// TwinCAT 3 PLC project Untitled1
// ProgramVersion: 3.1.4023.0
// libraries:
//   Tc2_EtherCAT, * (Beckhoff Automation GmbH)
//   Tc2_ModbusSrv, * (Beckhoff Automation GmbH)
//   Tc2_Standard, * (Beckhoff Automation GmbH)
//   Tc2_System, * (Beckhoff Automation GmbH)
//   Tc3_Module, * (Beckhoff Automation GmbH)
//   VisuDialogs, * (System)
//   BASIC,3.31,OSCAT
//   VisuSymbols,3.5.10.0,System
// project tree:
//   / Control.TcTTO, GlobalTextList.TcGTLO, Meter.TcTTO, PlcTask_1.TcTTO, Visualization Manager.TcVMO (not stored), VISU_TASK.TcTTO
//   DUTs/ CONVERTER.TcDUT
//   FUNC/ AVG_3.TcPOU, BYTE_UNION.TcPOU (not stored)
//   GVLs/ GVL_PM_CONFIG.TcGVL, GVL_GUI.TcGVL, GVL_HANDLER.TcGVL, GVL_POWERMETER.TcGVL, GVL_CONVERTERS_COMMON.TcGVL, GVL_CONV_COMMS.TcGVL, GVL_PLANT_DEF.TcGVL, GVL_P_CONTROL.TcGVL, GVL_Q_CONTROL.TcGVL, Meter_board_str.TcDUT
//   POUs/ BYTE_UNION.TcPOU, MAIN.TcPOU
//   POUs/CONTROL/ PI_BLOCK.TcPOU
//   POUs/CONVERTERS/ CONVERTERS_COMMS.TcPOU, Modbus_mapping.TcPOU, nN_coeff_calculation.TcPOU
//   POUs/EXTERNAL_COMMS/ Modbus_map.TcDUT
//   POUs/HANDLER_PARAM/ Data_transforming.TcPOU, Data_transform_float32.TcPOU, Data_transform_int64.TcPOU, MB_MAP_VARS_ENUM.TcTLEO, Parameters_handler.TcPOU, ReadWrite_Enum.TcDUT
//   POUs/METERING/ Analyzers.TcPOU, FB_EL3453_handling.TcPOU, METER_BOARD_CFG.TcPOU, METER_EL3453_CFG.TcPOU
//   POUs/P CONTROL/ Min_P_calculation.TcPOU, P_control_global.TcPOU, P_feedback_calculation.TcPOU
//   POUs/Q CONTROL/ Q_control_global.TcPOU, Q_ramp_module.TcPOU
//   POUs/VISU_HANDLER/ GUI_logic.TcPOU
//   VISUs/00_Main/ Main.TcVIS, Main_GUI.TcVIS
//   VISUs/01_P_control/ P_controller.TcVIS, P_min_indicator.TcTLO
//   VISUs/02_Q_control/ Q_controller.TcVIS
//   VISUs/03_Converters/ Conv_handling.TcVIS
//   VISUs/04_Powermeter/ M_board_status.TcTLO, PM_config.TcVIS
// real-time tasks:
//   TASK PlcTask: cycle T#5ms, priority 20, ADS port 350
//   TASK Control: cycle T#5ms, priority 1, ADS port 351
//   TASK Meter: cycle T#1ms, priority 2, ADS port 352
//   TASK VISU_TASK: cycle T#200000us, priority 30, ADS port 354
// I/O:
//   DEVICE Device 1 (EtherCAT) (disabled), AmsNetId 192.168.222.1.2.1
//     Term 1 (EK1200) [EK1200-7000 EtherCAT Power supply (1,5A E-Bus)] (disabled)
//       Term 4 (EL1259) [EL1259 8Ch. Dig Input 24V/8Ch. Dig. Output 24V with Multi-Time-Stamp] (disabled)
//       Term 5 (EL3453) [EL3453 3Ch. Power Measuring] (disabled)
//       Term 3 (EL9011) [EL9011 End Terminal]
// variable links:
//   Untitled1/Untitled1 Instance <-> Device 1 (EtherCAT)/Term 1 (EK1200)/Term 5 (EL3453)
//     Meter Inputs/GVL_POWERMETER.M_board_Freq_Hz <-> Total Basic/Frequency
//     Meter Inputs/GVL_POWERMETER.M_board_I_L1_angle <-> Total System Angles/Current Angle L1
//     Meter Inputs/GVL_POWERMETER.M_board_I_L2_angle <-> Total System Angles/Current Angle L2
//     Meter Inputs/GVL_POWERMETER.M_board_I_L3_angle <-> Total System Angles/Current Angle L3
//     Meter Inputs/GVL_POWERMETER.M_board_P_L1_kW <-> L1 Power/Active Power
//     Meter Inputs/GVL_POWERMETER.M_board_P_L2_kW <-> L2 Power/Active Power
//     Meter Inputs/GVL_POWERMETER.M_board_P_L3_kW <-> L3 Power/Active Power
//     Meter Inputs/GVL_POWERMETER.M_board_P_kW <-> Total Active Reduced/Active Power
//     Meter Inputs/GVL_POWERMETER.M_board_Q_L1_kVAr <-> L1 Power/Reactive Power
//     Meter Inputs/GVL_POWERMETER.M_board_Q_L2_kVAr <-> L2 Power/Reactive Power
//     Meter Inputs/GVL_POWERMETER.M_board_Q_L3_kVAr <-> L3 Power/Reactive Power
//     Meter Inputs/GVL_POWERMETER.M_board_Q_kVAr <-> Total Reactive Reduced/Reactive Power
//     Meter Inputs/GVL_POWERMETER.M_board_S_L1_kVA <-> L1 Power/Apparent Power
//     Meter Inputs/GVL_POWERMETER.M_board_S_L2_kVA <-> L2 Power/Apparent Power
//     Meter Inputs/GVL_POWERMETER.M_board_S_L3_kVA <-> L3 Power/Apparent Power
//     Meter Inputs/GVL_POWERMETER.M_board_S_kVA <-> Total Apparent Reduced/Apparent Power
//     Meter Inputs/GVL_POWERMETER.M_board_V_L1L2_Volt <-> Total L-L Voltages/L1-L2 Voltage
//     Meter Inputs/GVL_POWERMETER.M_board_V_L2L3_Volt <-> Total L-L Voltages/L2-L3 Voltage
//     Meter Inputs/GVL_POWERMETER.M_board_V_L3L1_Volt <-> Total L-L Voltages/L3-L1 Voltage
//     Meter Inputs/GVL_POWERMETER.M_board_V_L1L2_angle <-> Total System Angles/Voltage Angle L1L2
//     Meter Inputs/GVL_POWERMETER.M_board_V_L1L3_angle <-> Total System Angles/Voltage Angle L1L3
//     Meter Inputs/GVL_POWERMETER.M_board_V_L1N_Volt <-> L1 Basic/Voltage
//     Meter Inputs/GVL_POWERMETER.M_board_V_L2N_Volt <-> L2 Basic/Voltage
//     Meter Inputs/GVL_POWERMETER.M_board_V_L3N_Volt <-> L3 Basic/Voltage
//     Meter Inputs/GVL_POWERMETER.M_board_cos_phi <-> Total Basic/Power Factor
//     Meter Inputs/GVL_POWERMETER.M_board_cos_phi_L1 <-> L1 Power/Power Factor
//     Meter Inputs/GVL_POWERMETER.M_board_cos_phi_L2 <-> L2 Power/Power Factor
//     Meter Inputs/GVL_POWERMETER.M_board_cos_phi_L3 <-> L3 Power/Power Factor
//     PlcTask_1 Inputs/GVL_POWERMETER.M_board_Meter_status <-> InfoData/State

CONFIGURATION Untitled1
    RESOURCE PLC ON TwinCAT3
        TASK Control(INTERVAL := T#5ms, PRIORITY := 1);
        TASK Meter(INTERVAL := T#1ms, PRIORITY := 2);
        TASK PlcTask_1(INTERVAL := T#5ms, PRIORITY := 20);
        TASK VISU_TASK(INTERVAL := T#200000us, PRIORITY := 30);
        PROGRAM Q_control_global WITH Control : Q_control_global;
        PROGRAM P_control_global WITH Control : P_control_global;
        PROGRAM Analyzers WITH Meter : Analyzers;
        PROGRAM MAIN WITH PlcTask_1 : MAIN;
        PROGRAM VisuElems_Visu_Prg WITH VISU_TASK : VisuElems.Visu_Prg;
    END_RESOURCE
END_CONFIGURATION

// ---- DUTs/CONVERTER.TcDUT
TYPE CONVERTER :
STRUCT
	ReadRegs_INV: FB_MBReadRegs;
	WriteRegs_INV: FB_MBWriteRegs;
	
	Capacity: REAL:= 1000;				//Snominal from inverter in kVA
	IP: STRING(15):= '192.168.1.254';
	Port: UINT:= 502;					//Modbus port
	UnitID: BYTE:= 1;					//Modbus ID if necessary
	LengthRead: WORD:= 10;				//Amount of registers read from modbus
	LengthWrite: WORD:= 10;				//Amount of registers written via modbus
	InitAdressRead: WORD:= 7000;
	InitAdressWrite: WORD:= 8000;
	cbLenght: UDINT:= 2;
	READING: ARRAY [1..5] OF WORD;
    bReadBusy: BOOL;
    bReadError: BOOL;
    nReadErrorId: UDINT;
    nReadCount: UDINT;
	bWriteBusy: BOOL;
    bWriteError: BOOL;
    nWriteErrorId: UDINT;
    nWriteCount: UDINT;
	WRITING: ARRAY [1..7] OF WORD;
	ErrorCount: UDINT:= 0;
END_STRUCT
END_TYPE

// ---- GVLs/Meter_board_str.TcDUT
TYPE Meter_board_str :
STRUCT
	
	//Single-phase electrical parameters in engineering units
	P_L1_kW:			REAL;
	P_L2_kW:			REAL;
	P_L3_kW:			REAL;
	Q_L1_kVAr:			REAL;
	Q_L2_kVAr:			REAL;
	Q_L3_kVAr:			REAL;
	S_L1_kVA:			REAL;
	S_L2_kVA:			REAL;
	S_L3_kVA:			REAL;
	cos_phi_L1:			REAL;
	cos_phi_L2:			REAL;
	cos_phi_L3:			REAL;
	V_L1N_Volt:			REAL;
	V_L2N_Volt:			REAL;
	V_L3N_Volt:			REAL;

	//Three-phase electrical parameters in engineering units
	P_kW:				REAL;
	Q_kVAr:				REAL;
	S_kVA:				REAL;
	Freq_Hz:			REAL;
	cos_phi:			REAL;
	V_L1L2_Volt:		REAL;
	V_L2L3_Volt:		REAL;
	V_L3L1_Volt:		REAL;
	I_L1_angle:			REAL;
	I_L2_angle:			REAL;
	I_L3_angle:			REAL;
	V_L1L2_angle:		REAL;
	V_L1L3_angle:		REAL;
	
END_STRUCT
END_TYPE

// ---- POUs/EXTERNAL_COMMS/Modbus_map.TcDUT
{attribute 'qualified_only'}
{attribute 'strict'}
TYPE Modbus_map :
(
	enum_member := 0
);
END_TYPE

// ---- POUs/HANDLER_PARAM/MB_MAP_VARS_ENUM.TcTLEO
TYPE MB_MAP_VARS_ENUM :
(
	Plant_S_nom:= 0,
	Plant_V_nom:= 2,
	Plant_f_nom:= 4,
	N_converters:= 20,
	nN_converters:= 21,
	Control_conv_0:= 22,
	Control_conv_1:= 23,
	Control_conv_2:= 24,
	Control_conv_3:= 25,
	Control_conv_4:= 26,
	Control_conv_5:= 27,
	Control_conv_6:= 28,
	Control_conv_7:= 29,
	Control_conv_8:= 30,
	Control_conv_9:= 31,
	Control_conv_10:= 32,
	Control_conv_11:= 33,
	Control_conv_12:= 34,
	Control_conv_13:= 35,
	Control_conv_14:= 36,
	Control_conv_15:= 37,
	Control_conv_16:= 38,
	Control_conv_17:= 39,
	Control_conv_18:= 40,
	Control_conv_19:= 41,
	Control_conv_20:= 42,
	Control_conv_21:= 43,
	Control_conv_22:= 44,
	Control_conv_23:= 45,
	Control_conv_24:= 46,
	Control_conv_25:= 47,
	P_loop:= 300,
	P_reference:= 301,
	P_feedback:= 302,
	P_output:= 303,
	P_kp:= 304,
	P_kp_min:= 305,
	P_ti:= 306,
	P_high:= 307,
	P_low:= 308,
	P_invert:= 309,
	P_safety:= 310,
	P_min_charge:= 311,
	Q_loop:= 500,
	Q_reference:= 501,
	Q_feedback:= 502,
	Q_output:= 503,
	Q_kp:= 504,
	Q_kp_min:= 505,
	Q_ti:= 506,
	Q_high:= 507,
	Q_low:= 508,
	Q_invert:= 509,
	Q_safety:= 510,
	Ramp_enable:= 511,
	Time_span:= 512,
	R_up_value:= 513,
	R_down_value:= 514,
	R_units:= 515,
	P_L1_kW:= 1000,
	P_L2_kW:= 1002,
	P_L3_kW:= 1004,
	Q_L1_kVAr:= 1006,
	Q_L2_kVAr:= 1008,
	Q_L3_kVAr:= 1010,
	S_L1_kVA:= 1012,
	S_L2_kVA:= 1014,
	S_L3_kVA:= 1016,
	cos_phi_L1:= 1018,
	cos_phi_L2:= 1020,
	cos_phi_L3:= 1022,
	V_L1N_Volt:= 1024,
	V_L2N_Volt:= 1026,
	V_L3N_Volt:= 1028,
	P_tot_kW:= 1030,
	Q_tot_kVAr:= 1032,
	S_tot_kVA:= 1034,
	Freq_Hz:= 1036,
	cos_phi:= 1038,
	V_L1L2_Volt:= 1040,
	V_L2L3_Volt:= 1042,
	V_L3L1_Volt:= 1044,
	I_L1_angle:= 1046,
	I_L2_angle:= 1048,
	I_L3_angle:= 1050,
	V_L1L2_angle:= 1052,
	V_L1L3_angle:= 1054,
	V_phase_avg_Volt:= 1080,
	V_line_avg_Volt:= 1082,
	P_L1_pu:= 1084,
	P_L2_pu:= 1086,
	P_L3_pu:= 1088,
	Q_L1_pu:= 1090,
	Q_L2_pu:= 1092,
	Q_L3_pu:= 1094,
	S_L1_pu:= 1096,
	S_L2_pu:= 1098,
	S_L3_pu:= 1100,
	P_tot_pu:= 1102,
	Q_tot_pu:= 1104,
	S_tot_pu:= 1106,
	V_phase_avg_pu:= 1108,
	V_line_avg_pu:= 1110,
	Meter_status:= 1130,
	Lost_comms_enable:= 1131,
	Active_er_pos_kWh:= 1200,
	Active_er_neg_kWh:= 1204,
	Active_er_tot_kWh:= 1208,
	React_er_pos_kVArh:= 1212,
	React_er_neg_kVArh:= 1216,
	React_er_tot_kVArh:= 1220,
	Energies_reset:= 1224,
	V_ratio_RS:= 1300,
	V_ratio_ST:= 1302,
	V_ratio_TR:= 1304,
	I_ratio_R:=	1306,
	I_ratio_S:=	1308,
	I_ratio_T:=	1310

);
END_TYPE

// ---- POUs/HANDLER_PARAM/ReadWrite_Enum.TcDUT

TYPE ReadWrite_Enum :
(
	R_O := 0,
	R_W := 1
);
END_TYPE

// ---- GVLs/GVL_PM_CONFIG.TcGVL
{attribute 'qualified_only'}
VAR_GLOBAL
	
	//Variables needed to be in the data handling for the CoE analyzers boards configuration
	Device_Type_Index				: INT;
	Nominal_Voltage 				: REAL;
	Nominal_Frequency 				: REAL;
	Measurement_freq_range			: REAL;
	Current_trafo_dly_L1 			: REAL;			// Set variable for Current transformer delay L1	
	Current_trafo_dly_L2 			: REAL;			// Set variable for Current transformer delay L2
	Current_trafo_dly_L3 			: REAL;			// Set variable for Current transformer delay L3
	Current_trafo_range_L1 			: UDINT;		// Set variable for Current transformer range L1
	Current_trafo_range_L2 			: UDINT;		// Set variable for Current transformer range L2
	Current_trafo_range_L3 			: UDINT;		// Set variable for Current transformer range L3
	Voltage_Guard_Min_Error_L1		: REAL;			// Set variable for Voltage min error L1
	Voltage_Guard_Min_Error_L2		: REAL;			// Set variable for Voltage min error L2
	Voltage_Guard_Min_Error_L3		: REAL;			// Set variable for Voltage min error L3
	Voltage_Guard_Min_Warning_L1	: REAL;			// Set variable for Voltage min warning L1
	Voltage_Guard_Min_Warning_L2	: REAL;			// Set variable for Voltage min warning L2
	Voltage_Guard_Min_Warning_L3	: REAL;			// Set variable for Voltage min warning L3
	Voltage_Guard_Max_Warning_L1	: REAL;			// Set variable for Voltage max warning L1
	Voltage_Guard_Max_Warning_L2	: REAL;			// Set variable for Voltage max warning L2
	Voltage_Guard_Max_Warning_L3	: REAL;			// Set variable for Voltage max warning L3
	Voltage_Guard_Max_Error_L1		: REAL;			// Set variable for Voltage max error L1
	Voltage_Guard_Max_Error_L2		: REAL;			// Set variable for Voltage max error L2
	Voltage_Guard_Max_Error_L3		: REAL;			// Set variable for Voltage max error L3

	NetID_EL3XXX 		AT %I*	: AMSNETID ;
	SlaveID_EL3XXX 		AT %I*	: WORD ;
	 	
	NetID_EL3XXX_2 		AT %I*	: AMSNETID ;
	SlaveID_EL3XXX_2 	AT %I*	: WORD ;
END_VAR

VAR_GLOBAL PERSISTENT
	Current_trafo_rat_L1 			: REAL;			// Set variable for Current transformer ratio L1
	Current_trafo_rat_L2 			: REAL;			// Set variable for Current transformer ratio L2
	Current_trafo_rat_L3 			: REAL;			// Set variable for Current transformer ratio L3
	Voltage_trafo_rat_L1 			: REAL;			// Set variable for Voltage transformer ratio L1
	Voltage_trafo_rat_L2 			: REAL;			// Set variable for Voltage transformer ratio L2
	Voltage_trafo_rat_L3 			: REAL;			// Set variable for Voltage transformer ratio L3
END_VAR

// ---- GVLs/GVL_GUI.TcGVL
{attribute 'qualified_only'}
VAR_GLOBAL
	//Main GUI logic
	main_button_logic: 			BOOL:= TRUE;
	pcontrol_button_logic: 		BOOL:= FALSE;
	qcontrol_button_logic:		BOOL:= FALSE;
	conv_button_logic:			BOOL:= FALSE;
	meter_cfg_button_logic:		BOOL:= FALSE;
	
	frame_indic:				WORD:= 0;
	
	//P controller screen vars
	P_OL_sel_button:			BOOL:= FALSE;
	P_invert_button:			BOOL:= FALSE;
	
	//Q controller screen vars
	Q_OL_sel_button:			BOOL:= FALSE;
	Q_invert_button:			BOOL:= FALSE;
	
	//Converters screen
	Conv_online_button:			ARRAY [1..25] OF BOOL;
	Conv_on_off_button:			ARRAY [1..25] OF BOOL;
	Conv_n_mode_button:			ARRAY [1..25] OF BOOL;
END_VAR

// ---- GVLs/GVL_HANDLER.TcGVL
{attribute 'qualified_only'}
VAR_GLOBAL
	Init_vars:					BOOL; //initialization command
	Input_src:					bool:= false; //FALSE--> Via GUI, TRUE--> Via Modbus

	Modbus_srv_vars AT %MW0:	ARRAY [0..60000] OF WORD; //Variables for Modbus Server
	GUI_vars:					ARRAY [0..60000] OF REAL; //Variables for Web GUI
END_VAR

// ---- GVLs/GVL_POWERMETER.TcGVL
{attribute 'qualified_only'}
VAR_GLOBAL

	//Internal powermeter variables	
	Power_analyzer: 			Meter_board_str;
	Meter_comms_status: 		BOOL;
	
	//Internal calculated powermeter variables
		//Average voltages in engineering units
	V_phase_avg_Volt:			REAL;
	V_line_avg_Volt:			REAL;
		//Single-phase electrical parameters in p.u.
	P_L1_pu:					REAL;
	P_L2_pu:					REAL;
	P_L3_pu:					REAL;
	Q_L1_pu:					REAL;
	Q_L2_pu:					REAL;
	Q_L3_pu:					REAL;
	S_L1_pu:					REAL;
	S_L2_pu:					REAL;
	S_L3_pu:					REAL;
	V_L1N_pu:					REAL;
	V_L2N_pu:					REAL;
	V_L3N_pu:					REAL;
	I_L1_pu:					REAL;
	I_L2_pu:					REAL;
	I_L3_pu:					REAL;
		//Three-phase electrical parameters in p.u.
	P_pu:						REAL;
	Q_pu:						REAL;
	S_pu:						REAL;
		//Average voltages in engineering units
	V_phase_avg_pu:				REAL;
	V_line_avg_pu:				REAL;
	
	//Self-supply P variables
	P_min:						REAL; //Minimum P in p.u. of the system for PI feedback
	P_min_indicator:			WORD; //Minimum P indicator 0 --> L1; 1 --> L2; 2 --> L3

	//Enrgies handling & values
	Energies_reset:				BOOL:= FALSE;
	Active_er_neg_kWh: 			LINT:=0; //Active energy (three-phase) calculated if P_tot < 0
	Active_er_pos_kWh:			LINT:=0; //Active energy (three-phase) calculated if P_tot > 0
	Active_er_tot_kWh: 			LINT:=0; //Active energy (three-phase) calculated. Net calculation
	React_er_neg_kVArh: 		LINT:=0; //Rective energy (three-phase) calculated if Q_tot < 0
	React_er_pos_kVArh: 		LINT:=0; //Rective energy (three-phase) calculated if Q_tot > 0
	React_er_tot_kVArh: 		LINT:=0; //Reactive energy (three-phase) calculated. Net calculation
	
	//Data to be linked to metering board
	//Single-phase data
	M_board_P_L1_kW				AT %I*	: REAL;
	M_board_P_L2_kW				AT %I*	: REAL;		
	M_board_P_L3_kW				AT %I*	: REAL;		
	M_board_Q_L1_kVAr			AT %I*	: REAL;		
	M_board_Q_L2_kVAr			AT %I*	: REAL;		
	M_board_Q_L3_kVAr			AT %I*	: REAL;		
	M_board_S_L1_kVA			AT %I*	: REAL;		
	M_board_S_L2_kVA			AT %I*	: REAL;		
	M_board_S_L3_kVA			AT %I*	: REAL;		
	M_board_cos_phi_L1			AT %I*	: REAL;		
	M_board_cos_phi_L2			AT %I*	: REAL;		
	M_board_cos_phi_L3			AT %I*	: REAL;		
	M_board_V_L1N_Volt			AT %I*	: REAL;		
	M_board_V_L2N_Volt			AT %I*	: REAL;		
	M_board_V_L3N_Volt			AT %I*	: REAL;					
						
	//Three-phase data			
	M_board_P_kW				AT %I*	: REAL;	
	M_board_Q_kVAr				AT %I*	: REAL;	
	M_board_S_kVA				AT %I*	: REAL;	
	M_board_Freq_Hz				AT %I*	: REAL;		
	M_board_cos_phi				AT %I*	: REAL;		
	M_board_V_L1L2_Volt			AT %I*	: REAL;			
	M_board_V_L2L3_Volt			AT %I*	: REAL;			
	M_board_V_L3L1_Volt			AT %I*	: REAL;			
	M_board_I_L1_angle			AT %I*	: REAL;		
	M_board_I_L2_angle			AT %I*	: REAL;		
	M_board_I_L3_angle			AT %I*	: REAL;		
	M_board_V_L1L2_angle		AT %I* 	: REAL;			
	M_board_V_L1L3_angle		AT %I*	: REAL;					
	
	//Rest of data								
	M_board_Meter_status		AT %I*	: WORD;
	
	//Data from converters
	P_converters_tot:			REAL;
	Q_converters_tot:			REAL;
END_VAR

VAR_GLOBAL PERSISTENT
	Alg_lost_comms_enable: 		BOOL:= FALSE;
END_VAR

// ---- GVLs/GVL_CONVERTERS_COMMON.TcGVL
{attribute 'qualified_only'}
VAR_GLOBAL
	CONVERTER_STATUS_RUN:	WORD:= 1; //Status told by the inverter when injecting P and Q
END_VAR

// ---- GVLs/GVL_CONV_COMMS.TcGVL
{attribute 'qualified_only'}
VAR_GLOBAL
	// Variables written to converters
	Setpoint_P:			ARRAY [1..15] OF WORD; //P setpoint to converters in percentage
	Setpoint_Q:			ARRAY [1..15] OF INT; //Q setpoint to converters in percentage
	Start_Command:		ARRAY [1..15] OF BOOL; //Command to start (1) / stop (0) converters
	Night_Mode_Active: 	ARRAY [1..15] OF BOOL; //Command to activate (1) / deactivate (0) converter's night mode
	Watchdog_PPC: 		WORD := 1;			// Watchdog of PPC to warn comms
	
	// Variables read from converters
	P_Measured:			ARRAY [1..15] OF WORD; //P measured from converters in kW
	Q_Measured:			ARRAY [1..15] OF WORD; //Q measured from converters in kVAR
	S_Measured:			ARRAY [1..15] OF WORD; //S measured from converters in kVA
	cosphi_Measured:	ARRAY [1..15] OF WORD;
	Current_Status:		ARRAY [1..15] OF WORD; //Status told by the converter. Check converter's main FSM
	
	// Comms variables
	Error_task:			ARRAY [1..15] OF WORD; //converter under comms error (offline)
	Control_Byte: 		ARRAY [1..15] OF BYTE;
	Status_Byte: 		ARRAY [1..15] OF BYTE;
	
	//Rest of variables
	converters_nN_coeff:	REAL:= 1; //Coefficient that expresses amount of converters running over total
END_VAR

VAR_GLOBAL PERSISTENT
	//Converters definitions
	NUMBER_CONVERTERS: 	WORD:= 1; //Amount of conveters to control
	CONVERTERS:			ARRAY [1..15] OF CONVERTER;

	//Variables written to converters
	Comms_Control_Word:	ARRAY [1..15] OF WORD; //Word to summarize bitwisely commands to converters
END_VAR

// ---- GVLs/GVL_PLANT_DEF.TcGVL
{attribute 'qualified_only'}
VAR_GLOBAL PERSISTENT
	Plant_capacity_nom:			REAL:= 4000; //Total capacity in kVA
	PoC_Voltage_nom:			REAL:= 20000;//Point of Connection voltage in V
	PoC_freq_nom:				REAL:= 50; //Point of Connection frequency in Hz
	
	dummy:WORD:=0;
	switch_col:BOOL;
END_VAR

// ---- GVLs/GVL_P_CONTROL.TcGVL
{attribute 'qualified_only'}
VAR_GLOBAL
	//Control and PI variables
	P_feedback:		REAL:= 1; //Feedback for PI control
	P_output:		REAL:= 1; //Output of P control block	

	//Control and PI variables
	P_err_signal:	REAL:= 0; //Error signal calculated in PI´
END_VAR

VAR_GLOBAL PERSISTENT
	P_loop_type:	BOOL:= 0; //0 --> Control in CL; 1 --> Control in OL.
	
	//Control and PI variables
	P_reference:	REAL:= 0.02; //Input of P control block	
	P_kp:			REAL:= 0.05; //Kp for P control
	P_kp_min:		REAL:= 0.05; //Kp minimum for P control
	P_Ti:			REAL:= 2; //Ti for P control
	P_high_act:		REAL:= 100; //P high for PI antiwind up. Max control action
	P_low_act:		REAL:= 0; //P low for PI antiwind up. Min control action
	P_invert:		BOOL:= FALSE; //PI inversion
	
	//Safety position
	P_safety:		REAL:= 0; //P setpoint to converters at safety position
END_VAR

// ---- GVLs/GVL_Q_CONTROL.TcGVL
{attribute 'qualified_only'}
VAR_GLOBAL
	
	//Control and PI variables
	Q_feedback:			REAL:= 1; //Feedback for PI control
	Q_output:			REAL:= 1; //Output of Q control block
	Q_err_signal:		REAL:= 0; //Error signal calculated in PI´
	
	Time_span:			REAL:= 60; //Time length in s of ramp action
END_VAR

VAR_GLOBAL PERSISTENT
	Q_loop_type:		BOOL:= 1; //0 --> Control in CL; 1 --> Control in OL.

	//Control and PI variables
	Q_reference:		REAL:= 0; //Input of Q control block
	Q_kp:				REAL:= 0.05; //Kp for Q control
	Q_kp_min:			REAL:= 0.05; //Kp minimum for Q control
	Q_Ti:				REAL:= 3; //Ti for Q control
	Q_high_act:			REAL:= 100; //Q high for PI antiwind up. Max control action
	Q_low_act:			REAL:= -100; //Q low for PI antiwind up. Min control action
	Q_invert:			BOOL:= FALSE; //PI inversion
	
	//Safety position
	Q_safety:			REAL:= 0; //Q setpoint to converters at safety position
	
	//Ramps module
	Ramp_enable:		BOOL:= FALSE; //Ramp functionality enable
	Ramp_up_value:		REAL; //Increasing ramp value (units depend on selector)
	Ramp_down_value:	REAL; //Increasing ramp value (units depend on selector)
	Ramp_units:			WORD; //0 --> Ramp in %/s; 1 --> %/min; 2 --> %/h
END_VAR

// ---- POUs/Q CONTROL/Q_control_global.TcPOU
PROGRAM Q_control_global
VAR
	//Functions to be called
	PI_Q:			PI_BLOCK;
	Q_Ramp:			Q_ramp_module;
	
	//Control varaibles
	Q_setpoint:		REAL;
	Q_feedback:		real;
END_VAR

//Control variables assignment
Q_setpoint:= GVL_Q_CONTROL.Q_reference;
Q_feedback:= GVL_POWERMETER.Q_pu;

IF GVL_Q_CONTROL.Ramp_enable THEN

	Q_Ramp(
		Q_reference:= Q_setpoint, 
		Ramp_increasing_val:= GVL_Q_CONTROL.Ramp_up_value, 
		Ramp_decreasing_val:= GVL_Q_CONTROL.Ramp_down_value, 
		Ramp_unit_sel:= GVL_Q_CONTROL.Ramp_units, 
		Q_ramp_out=> Q_setpoint,
		Time_span=> GVL_Q_CONTROL.Time_span);
END_IF

IF GVL_Q_CONTROL.Q_loop_type THEN
	//Open loop control case
	GVL_Q_CONTROL.Q_output:= Q_setpoint;
ELSE
	//Closed loop control case
	PI_Q(
		Setpoint:= Q_setpoint, 
		Feedback:= Q_feedback, 
		Inverted_PID:= GVL_Q_CONTROL.Q_invert, 
		KP:= GVL_Q_CONTROL.Q_kp, 
		KP_Min:= GVL_Q_CONTROL.Q_kp_min, 
		TI:= GVL_Q_CONTROL.Q_Ti, 
		Antiwindup_max:= GVL_Q_CONTROL.Q_high_act, 
		Antiwindup_min:= GVL_Q_CONTROL.Q_low_act, 
		Output_prev:= GVL_Q_CONTROL.Q_output, 
		Output=> GVL_Q_CONTROL.Q_output, 
		Error_Out=> GVL_Q_CONTROL.Q_err_signal);
END_IF

END_PROGRAM

// ---- POUs/CONTROL/PI_BLOCK.TcPOU
FUNCTION_BLOCK PI_BLOCK
VAR_INPUT
	Setpoint: REAL;
	Feedback: REAL;
	
	Inverted_PID: BOOL := 0;
	KP: REAL;
	KP_Min: REAL;
	TI: REAL;
	
	Antiwindup_max: REAL;
	Antiwindup_min: REAL;
	Output_prev: REAL;
END_VAR
VAR_OUTPUT
	Output: REAL;
	Error_Out: REAL;
END_VAR
VAR
	Error: REAL;
	Ki: REAL;
	I_filtered: REAL;
	KP_Operator: REAL;
	kp_minimum: REAL;
END_VAR

(*
 ************************************************************************************************************
 * \file  PI_BLOCK
 * \author Quique
 * \version 1.0.0
 * \Date Creation: 19/06/2022
 * \brief PI function used for closed loop controls
 ************************************************************************************************************
 \defgroup CONTROL
 
 \brief 	This block implements a PI to control electrical variables in closed loop (P and Q)
		
 \details 	First part considers if PI is configured to be inverter and calculates error signal
 			
 			Second part calculates integral action and applies antiwindup on it to guarantee integral action
			by itself doesn't reach extremely high levels. It's also relevant to highlight that integral 
			action is calculated using pervious output. Thus, this PI is suitable for all sampling times
			(It doesn`t requires user to input it) and it can be easy de-saturated when needed.
			
			Third part calculates proportional action dinamically. It means, there are 2 defined KPs, so
			that depending on the error signal calculated the greater the error, the greater the KP (nearer
			to Kp value) and if the error is low, proportional action will be near to Kp_min. If user doesn't
			want this functionality, it is enough equaling Kp and Kp_min.
			
			Fourth section inverts PI if needed.
			
			Fifth section applies antiwindup limits to the output calculated.
 
*)
 
//Error calculation part         
IF Inverted_PID THEN;
	Error := Feedback - Setpoint;
ELSE
	Error := Setpoint - Feedback;
END_IF
Error_Out := Error;

//Integral action calculation
IF TI > 0 THEN
	Ki := 1 / TI;
ELSE
	Ki := 0;
END_IF	
I_filtered := (I_filtered + ((Output_prev - I_filtered) * Ki));

//Antiwindup calculation and usage on output
IF (I_filtered >= Antiwindup_max) THEN;
	I_filtered := Antiwindup_max;
ELSIF (I_filtered <= Antiwindup_min) THEN;
	I_filtered := Antiwindup_min;
END_IF

//Proportional action calculation
kp_minimum:= MIN(KP_Min, KP);

KP_Operator := (ABS(KP - KP_Min) * ABS(Error)) + kp_minimum;
KP_Operator := ABS(KP_Operator);

//PI output calculation - Control action calculation
Output := I_filtered + KP_Operator * (Setpoint - Feedback);

//PI inversion if applied
IF Inverted_PID = 1 THEN;
	Output := - Output;
END_IF

//Antiwindup calculation and usage on output
IF (Output >= Antiwindup_max) THEN;
	Output := Antiwindup_max;
ELSIF (Output <= Antiwindup_min) THEN;
	Output := Antiwindup_min;
END_IF

END_FUNCTION_BLOCK

// ---- POUs/Q CONTROL/Q_ramp_module.TcPOU
FUNCTION_BLOCK Q_ramp_module
VAR_INPUT
	Q_reference: 				REAL;
	Ramp_increasing_val: 		REAL;
	Ramp_decreasing_val: 		REAL;
	Ramp_unit_sel:				WORD;
END_VAR

VAR_OUTPUT
	Q_ramp_out: 				REAL;
	Time_span: 					REAL;
END_VAR

VAR
	First_Iterarion: 			BOOL:= FALSE;
	Q_error: 					REAL;
	Aux_ramp: 					REAL;
	Lim_ramp: 					REAL;
	Ref_Prev: 					REAL;
	
	Ramp_scaled: 				REAL;	
	Ramp_aux_scaled: 			REAL;
	Ramp_incr_scaled: 			REAL;
	Ramp_decr_scaled: 			REAL;

	Executing_time:  			REAL:= 0.005; //Time of task execution
END_VAR

CASE Ramp_unit_sel OF
	0: //Ramp in %/s
		Time_span:= 1;
	1: //Ramp in %/min
		Time_span:= 60;
	2:	//Ramp in %/h
		Time_span:= 3600;
END_CASE

IF GVL_Q_CONTROL.Ramp_enable THEN	
	//Inicialization of the ramp to the measurement
	IF First_Iterarion THEN
		
		Ref_prev:= GVL_POWERMETER.Q_pu; 
		First_Iterarion := FALSE;
	
	END_IF
	
	IF Q_ramp_out <> Q_reference THEN
		
		// First of all, calculate the error of Q
		Q_error:= Q_reference - Ref_Prev;
			
		//Aux slope calculation and Slopes escalation:
		Ramp_aux_scaled:= Q_error / Executing_time; 
		Ramp_incr_scaled:= Ramp_increasing_val/Time_span;
		Ramp_decr_scaled:= Ramp_decreasing_val/Time_span;
	
		//Limiting the ramp
		Lim_ramp:= LIMIT(Ramp_decr_scaled, Ramp_aux_scaled, Ramp_incr_scaled);
		
		//Output
		Ramp_scaled:= Lim_ramp;
		Q_ramp_out:= (Ramp_scaled * Executing_time) + Ref_Prev;
		Ref_Prev:= Q_ramp_out;
	END_IF
END_IF

END_FUNCTION_BLOCK

// ---- POUs/P CONTROL/P_control_global.TcPOU
PROGRAM P_control_global
VAR
	P_PI: PI_BLOCK;
END_VAR

P_feedback_calculation();

IF GVL_P_CONTROL.P_loop_type THEN
	//Open loop control case
	GVL_P_CONTROL.P_output:= GVL_P_CONTROL.P_reference;
ELSE
	//Closed loop control case
	P_PI(
		Setpoint:= GVL_P_CONTROL.P_reference, 
		Feedback:= GVL_P_CONTROL.P_feedback, 
		Inverted_PID:= GVL_P_CONTROL.P_invert, 
		KP:= GVL_P_CONTROL.P_kp, 
		KP_Min:= GVL_P_CONTROL.P_kp_min, 
		TI:= GVL_P_CONTROL.P_Ti, 
		Antiwindup_max:= GVL_P_CONTROL.P_high_act, 
		Antiwindup_min:= GVL_P_CONTROL.P_low_act, 
		Output_prev:= GVL_P_CONTROL.P_output, 
		Output=> GVL_P_CONTROL.P_output, 
		Error_Out=> GVL_P_CONTROL.P_err_signal);
END_IF

END_PROGRAM

// ---- POUs/P CONTROL/P_feedback_calculation.TcPOU
PROGRAM P_feedback_calculation
VAR
END_VAR

(*
 *************************************************************************************************************
 * \file  P_feedback_calc
 * \author Quique
 * \version 1.0.0
 * \date Creation: 16/07/2021
 * \brief Selects P used in feedback 
 *************************************************************************************************************
 \defgroup P_CONTROL - FEEDBACK_CALC
 
 \brief 	This algorithm is used to determine which is the phase with the less power consumption and then
 			this obtained value is used as the feedback of P loop. The goal is that this value
			is updated continuously to guarantee that there is null P injection to grid during stationary
			regime. 
		
 \details 	This algorithm is based on a first order approach assuming that line power equals the summatory 
			of 3 single - phase powers. Thus and since it is mandatory to not inject P to grid, the algorithm
			checks which is the phase with the less consumption value, multiplies it by three 

*)

//Determination of P_measured_min
Min_P_calculation();

//  Ploop in closed loop
IF NOT GVL_P_CONTROL.P_loop_type THEN
	GVL_P_CONTROL.P_feedback:= GVL_POWERMETER.P_min;
ELSE
// Ploop in open loop	
	GVL_P_CONTROL.P_feedback:= GVL_POWERMETER.P_pu;
END_IF

END_PROGRAM

// ---- POUs/P CONTROL/Min_P_calculation.TcPOU
PROGRAM Min_P_calculation
VAR
	P_L1_ABS: REAL;
	P_L2_ABS: REAL;
	P_L3_ABS: REAL;
	
	P_L1_pu: REAL;
	P_L2_pu: REAL;
	P_L3_pu: REAL;
	
	P_min_indic: WORD:= 0;
	P_min_pu: REAL:= 0;
	P_min_3ph: REAL;
	
END_VAR

(*
 *************************************************************************************************************
 * \file  Min_P_calculation
 * \author Quique
 * \version 1.0.0
 * \date Creation: 16/07/2022
 * \brief Determines which is the minimal P for P CL
 *************************************************************************************************************
 \defgroup P_CONTROLS - MIN_P_CALCULATION
 
 \brief 	This algorithm is used to determine which is the phase with the less power consumption and then
 			this obtained value is used as the feedback of P loop of the system. The goal is that this value
			is updated continuously to guarantee that there is null P injection to grid during stationary
			regime, according to RD 244/19. 
		
 \details 	It is based on a first order approach assuming that line power equals the summatory 
			of 3 single - phase powers (it assumes system loads are balanced. Thus and as it is mandatory
			not to inject P to grid, the algorithm checks which is the single - phase power with the less 
			consumption value, multiplies it by three and then it takes that value as P closed loop feedback, 
			to have closed loop working in a pseudo three-phase, since all inverters generate 3-phase
			balanced current, for P PI.
			
			In Open Loop it is not considered, since OL control doesn´t meet RD 244/19 requirements.

*)
	
//P_meas min determination
P_L1_ABS:= ABS(GVL_POWERMETER.Power_analyzer.P_L1_kW);
P_L2_ABS:= ABS(GVL_POWERMETER.Power_analyzer.P_L2_kW);
P_L3_ABS:= ABS(GVL_POWERMETER.Power_analyzer.P_L3_kW);

IF (P_L1_ABS < P_L2_ABS) AND (P_L1_ABS < P_L3_ABS) THEN
	P_min_indic:= 0;
ELSIF (P_L2_ABS < P_L1_ABS) AND (P_L2_ABS < P_L3_ABS) THEN
	P_min_indic:= 1;
ELSE
	P_min_indic:= 2;
END_IF

//P_measured single-phase in p.u. 
P_L1_pu:= GVL_POWERMETER.P_L1_pu;
P_L2_pu:= GVL_POWERMETER.P_L2_pu;
P_L3_pu:= GVL_POWERMETER.P_L3_pu;

//P_meas_min selection
P_min_pu:= MUX(P_min_indic, P_L1_pu, P_L2_pu, P_L3_pu);
GVL_POWERMETER.P_min_indicator:= P_min_indic;

//feedback value
P_min_3ph:= P_min_pu * 3;
GVL_POWERMETER.P_min:= P_min_3ph;

END_PROGRAM

// ---- POUs/METERING/Analyzers.TcPOU
PROGRAM Analyzers
VAR
	PM_beck_EL3453:			FB_EL3453_handling;
	
	S_nom_facility_inv:			REAL; //Inverse of Snom [1/kVA]
	V_nom_facility_inv:			REAL; //Inverse of Snom [1/V]
	
	P_inverters:				REAL:= 0; //Sum of Pread from all inverters
	Q_inverters:				REAL:= 0; //Sum of Qread from all inverters
	i:							WORD:= 1;
END_VAR

VAR CONSTANT
	tick_hourly: 				REAL:= 2.78E-7; //ms expressed in hours (how much hours is a tick)
END_VAR


PM_beck_EL3453(Analyzer_str_out=> GVL_POWERMETER.Power_analyzer);

//Average voltages obtention
GVL_POWERMETER.V_phase_avg_Volt:= AVG_3(GVL_POWERMETER.Power_analyzer.V_L1N_Volt, 
										GVL_POWERMETER.Power_analyzer.V_L2N_Volt, 
										GVL_POWERMETER.Power_analyzer.V_L3N_Volt);
										
GVL_POWERMETER.V_line_avg_Volt:= AVG_3(GVL_POWERMETER.Power_analyzer.V_L1L2_Volt, 
										GVL_POWERMETER.Power_analyzer.V_L2L3_Volt, 
										GVL_POWERMETER.Power_analyzer.V_L3L1_Volt);

//Basis for per unit calculations
IF GVL_PLANT_DEF.Plant_capacity_nom <= 0 THEN
	S_nom_facility_inv:= 0;
ELSE
	S_nom_facility_inv:= 1 / GVL_PLANT_DEF.Plant_capacity_nom;
END_IF

//Per unit values obtention - Single-phase powers
GVL_POWERMETER.P_L1_pu:= GVL_POWERMETER.Power_analyzer.P_L1_kW * S_nom_facility_inv;
GVL_POWERMETER.P_L2_pu:= GVL_POWERMETER.Power_analyzer.P_L2_kW * S_nom_facility_inv;
GVL_POWERMETER.P_L3_pu:= GVL_POWERMETER.Power_analyzer.P_L3_kW * S_nom_facility_inv;
GVL_POWERMETER.Q_L1_pu:= GVL_POWERMETER.Power_analyzer.Q_L1_kVAr * S_nom_facility_inv;
GVL_POWERMETER.Q_L2_pu:= GVL_POWERMETER.Power_analyzer.Q_L2_kVAr * S_nom_facility_inv;
GVL_POWERMETER.Q_L3_pu:= GVL_POWERMETER.Power_analyzer.Q_L3_kVAr * S_nom_facility_inv;
GVL_POWERMETER.S_L1_pu:= GVL_POWERMETER.Power_analyzer.S_L1_kVA * S_nom_facility_inv;
GVL_POWERMETER.S_L2_pu:= GVL_POWERMETER.Power_analyzer.S_L2_kVA * S_nom_facility_inv;
GVL_POWERMETER.S_L3_pu:= GVL_POWERMETER.Power_analyzer.S_L3_kVA * S_nom_facility_inv;

//Per unit values obtention - Three-phase powers
GVL_POWERMETER.P_pu:= GVL_POWERMETER.Power_analyzer.P_kW * S_nom_facility_inv;
GVL_POWERMETER.Q_pu:= GVL_POWERMETER.Power_analyzer.Q_kVAr * S_nom_facility_inv;
GVL_POWERMETER.S_pu:= GVL_POWERMETER.Power_analyzer.S_kVA * S_nom_facility_inv;

//Per unit values obtention - Voltages
GVL_POWERMETER.V_line_avg_pu:= GVL_POWERMETER.V_line_avg_Volt * V_nom_facility_inv;
GVL_POWERMETER.V_phase_avg_pu:= GVL_POWERMETER.V_phase_avg_Volt * V_nom_facility_inv;

IF GVL_POWERMETER.V_phase_avg_pu <> 0 THEN
	GVL_POWERMETER.V_L1N_pu:= GVL_POWERMETER.Power_analyzer.V_L1N_Volt / GVL_POWERMETER.V_phase_avg_pu;
	GVL_POWERMETER.V_L2N_pu:= GVL_POWERMETER.Power_analyzer.V_L2N_Volt / GVL_POWERMETER.V_phase_avg_pu;
	GVL_POWERMETER.V_L3N_pu:= GVL_POWERMETER.Power_analyzer.V_L3N_Volt / GVL_POWERMETER.V_phase_avg_pu;
END_IF
	
//Per unit currents obtention
IF (GVL_POWERMETER.V_L1N_pu <> 0) AND (GVL_POWERMETER.Power_analyzer.cos_phi_L1 <> 0) THEN
	GVL_POWERMETER.I_L1_pu:= GVL_POWERMETER.P_L1_pu / (GVL_POWERMETER.V_L1N_pu * GVL_POWERMETER.Power_analyzer.cos_phi_L1);
END_IF
IF (GVL_POWERMETER.V_L2N_pu <> 0) AND (GVL_POWERMETER.Power_analyzer.cos_phi_L2 <> 0) THEN
	GVL_POWERMETER.I_L2_pu:= GVL_POWERMETER.P_L2_pu / (GVL_POWERMETER.V_L2N_pu * GVL_POWERMETER.Power_analyzer.cos_phi_L2);
END_IF
IF (GVL_POWERMETER.V_L3N_pu <> 0) AND (GVL_POWERMETER.Power_analyzer.cos_phi_L3 <> 0) THEN
	GVL_POWERMETER.I_L3_pu:= GVL_POWERMETER.P_L3_pu / (GVL_POWERMETER.V_L3N_pu * GVL_POWERMETER.Power_analyzer.cos_phi_L3);
END_IF
	
//Active energies calculation. It is an infinitesimal addition (an integration of P_measured)
GVL_POWERMETER.Active_er_tot_kWh:= REAL_TO_LINT(GVL_POWERMETER.Power_analyzer.P_kW * tick_hourly) + 
												GVL_POWERMETER.Active_er_tot_kWh;
IF GVL_POWERMETER.Power_analyzer.P_kW  >= 0 THEN
	GVL_POWERMETER.Active_er_pos_kWh:= REAL_TO_LINT(GVL_POWERMETER.Power_analyzer.P_kW * tick_hourly) + 
													GVL_POWERMETER.Active_er_pos_kWh;
ELSE	
	GVL_POWERMETER.Active_er_neg_kWh:= REAL_TO_LINT(GVL_POWERMETER.Power_analyzer.P_kW * tick_hourly) + 
													GVL_POWERMETER.Active_er_neg_kWh;
END_IF
	
//Reactive energies calculation. It is an infinitesimal addition (an integration of Q_measured)
GVL_POWERMETER.React_er_tot_kVArh:= REAL_TO_LINT(GVL_POWERMETER.Power_analyzer.Q_kVAr * tick_hourly) + 
												GVL_POWERMETER.React_er_tot_kVArh;
IF GVL_POWERMETER.Power_analyzer.Q_kVAr >= 0 THEN
	GVL_POWERMETER.React_er_pos_kVArh:= REAL_TO_LINT(GVL_POWERMETER.Power_analyzer.Q_kVAr * tick_hourly) + 
													GVL_POWERMETER.React_er_pos_kVArh;
ELSE
	GVL_POWERMETER.React_er_neg_kVArh:= REAL_TO_LINT(GVL_POWERMETER.Power_analyzer.Q_kVAr * tick_hourly) + 
													GVL_POWERMETER.React_er_neg_kVArh;
END_IF

//Energies reset when desired
IF GVL_POWERMETER.Energies_reset THEN
	GVL_POWERMETER.Active_er_neg_kWh:= 0;
	GVL_POWERMETER.Active_er_pos_kWh:= 0;
	GVL_POWERMETER.Active_er_tot_kWh:= 0;
	GVL_POWERMETER.React_er_neg_kVArh:= 0;
	GVL_POWERMETER.React_er_pos_kVArh:= 0;
	GVL_POWERMETER.React_er_tot_kVArh:= 0;
	
	GVL_POWERMETER.Energies_reset:= FALSE;
END_IF

//Powermeter variables publishing via Modbus
MEMCPY(destAddr:= ADR(GVL_HANDLER.Modbus_srv_vars[P_L1_kW]), srcAddr:= ADR(GVL_POWERMETER.Power_analyzer), n:= SIZEOF(GVL_POWERMETER.Power_analyzer));
		
//Config calling
METER_BOARD_CFG();

//Addition of P and Q from inverters
FOR i:=1 TO GVL_CONV_COMMS.NUMBER_CONVERTERS DO;
	P_inverters:= P_inverters + GVL_CONV_COMMS.P_Measured[i];
	Q_inverters:= Q_inverters + GVL_CONV_COMMS.Q_Measured[i];
END_FOR

GVL_POWERMETER.P_converters_tot:= P_inverters;
GVL_POWERMETER.Q_converters_tot:= Q_inverters;
P_inverters:= 0;
Q_inverters:= 0;

END_PROGRAM

// ---- POUs/METERING/FB_EL3453_handling.TcPOU
FUNCTION_BLOCK FB_EL3453_handling
VAR_INPUT
END_VAR

VAR_OUTPUT
	Analyzer_str_out:			Meter_board_str;
END_VAR

VAR
END_VAR

VAR CONSTANT
	CTE_1E_M3:					REAL:= 0.001;
END_VAR

//Single-phase powers linkage + structure writing and scaling
Analyzer_str_out.P_L1_kW:= GVL_POWERMETER.M_board_P_L1_kW * CTE_1E_M3;
Analyzer_str_out.P_L2_kW:= GVL_POWERMETER.M_board_P_L2_kW * CTE_1E_M3;
Analyzer_str_out.P_L3_kW:= GVL_POWERMETER.M_board_P_L3_kW * CTE_1E_M3;
Analyzer_str_out.Q_L1_kVAr:= GVL_POWERMETER.M_board_Q_L1_kVAr * CTE_1E_M3;
Analyzer_str_out.Q_L2_kVAr:= GVL_POWERMETER.M_board_Q_L2_kVAr * CTE_1E_M3;
Analyzer_str_out.Q_L3_kVAr:= GVL_POWERMETER.M_board_Q_L3_kVAr * CTE_1E_M3;
Analyzer_str_out.S_L1_kVA:= GVL_POWERMETER.M_board_S_L1_kVA * CTE_1E_M3;
Analyzer_str_out.S_L2_kVA:= GVL_POWERMETER.M_board_S_L2_kVA * CTE_1E_M3;
Analyzer_str_out.S_L3_kVA:= GVL_POWERMETER.M_board_S_L3_kVA * CTE_1E_M3;

//Single-phase cos(phi) + structure writing 
Analyzer_str_out.cos_phi_L1:= GVL_POWERMETER.M_board_cos_phi_L1;
Analyzer_str_out.cos_phi_L2:= GVL_POWERMETER.M_board_cos_phi_L2;
Analyzer_str_out.cos_phi_L3:= GVL_POWERMETER.M_board_cos_phi_L3;

//Phase voltages + structure writing 
Analyzer_str_out.V_L1N_Volt:= GVL_POWERMETER.M_board_V_L1N_Volt;
Analyzer_str_out.V_L2N_Volt:= GVL_POWERMETER.M_board_V_L2N_Volt;
Analyzer_str_out.V_L3N_Volt:= GVL_POWERMETER.M_board_V_L3N_Volt;

//Three-phase powers linkage + structure writing and scaling
Analyzer_str_out.P_kW:= GVL_POWERMETER.M_board_P_kW * CTE_1E_M3;
Analyzer_str_out.Q_kVAr:= GVL_POWERMETER.M_board_Q_kVAr * CTE_1E_M3;
Analyzer_str_out.S_kVA:= GVL_POWERMETER.M_board_S_kVA * CTE_1E_M3;

//Line voltages + structure writing 
Analyzer_str_out.V_L1L2_Volt:= GVL_POWERMETER.M_board_V_L1L2_Volt;
Analyzer_str_out.V_L2L3_Volt:= GVL_POWERMETER.M_board_V_L2L3_Volt;
Analyzer_str_out.V_L3L1_Volt:= GVL_POWERMETER.M_board_V_L3L1_Volt;

//System angles
Analyzer_str_out.I_L1_angle:= GVL_POWERMETER.M_board_I_L1_angle;
Analyzer_str_out.I_L2_angle:= GVL_POWERMETER.M_board_I_L2_angle;
Analyzer_str_out.I_L3_angle:= GVL_POWERMETER.M_board_I_L3_angle;
Analyzer_str_out.V_L1L2_angle:= GVL_POWERMETER.M_board_V_L1L2_angle;
Analyzer_str_out.V_L1L3_angle:= GVL_POWERMETER.M_board_V_L1L3_angle;

//Rest of electrical parameters + structure writing 
Analyzer_str_out.Freq_Hz:= GVL_POWERMETER.M_board_Freq_Hz;
Analyzer_str_out.cos_phi:= GVL_POWERMETER.M_board_cos_phi;

END_FUNCTION_BLOCK

// ---- FUNC/AVG_3.TcPOU
FUNCTION AVG_3 : real
VAR_INPUT
	IN_1:			REAL;
	IN_2:			REAL;
	IN_3:			REAL;
END_VAR
VAR
	CTE_1_THIRD:	REAL:= 0.333333333333333333333;
END_VAR

AVG_3:= (IN_1 + IN_2 + IN_3) * CTE_1_THIRD;

END_FUNCTION

// ---- POUs/METERING/METER_BOARD_CFG.TcPOU
PROGRAM METER_BOARD_CFG
VAR
	
	Device_Type_Index : UINT:= 0;
	Device_Type : STRING;
	
	EL3XXX_Conf : METER_EL3453_CFG;
	Error_Selection: BOOL;
	Error_Nom_voltage : BOOL;
	Error_Nominal_Frequency : BOOL;				// Error read/writing nominal frequency
	Error_Measurement_freq_range : BOOL;		// Error read/writing frequency range working
	Error_Current_trafo_rat_L1 : BOOL;			// Error read/writing Current transformer ratio L1
	Error_Current_trafo_rat_L2 : BOOL;			// Error read/writing Current transformer ratio L2
	Error_Current_trafo_rat_L3 : BOOL;			// Error read/writing Current transformer ratio L3
	Error_Voltage_trafo_rat_L1 : BOOL;			// Error read/writing Voltage transformer ratio L1
	Error_Voltage_trafo_rat_L2 : BOOL;			// Error read/writing Voltage transformer ratio L2
	Error_Voltage_trafo_rat_L3 : BOOL;			// Error read/writing Voltage transformer ratio L3
	Error_Current_trafo_dly_L1 : BOOL;			// Error read/writing Current transformer delay L1	
	Error_Current_trafo_dly_L2 : BOOL;			// Error read/writing Current transformer delay L2
	Error_Current_trafo_dly_L3 : BOOL;			// Error read/writing Current transformer delay L3
	Error_Current_trafo_range_L1 : BOOL;		// Error read/writing Current transformer delay L1	
	Error_Current_trafo_range_L2 : BOOL;		// Error read/writing Current transformer delay L2
	Error_Current_trafo_range_L3 : BOOL;		// Error read/writing Current transformer delay L3
	Error_Voltage_Guard_Min_Error_L1: BOOL;		// Error read/writing Voltage min error L1
	Error_Voltage_Guard_Min_Error_L2: BOOL;		// Error read/writing Voltage min error L2
	Error_Voltage_Guard_Min_Error_L3: BOOL;		// Error read/writing Voltage min error L3
	Error_Voltage_Guard_Min_Warning_L1: BOOL;	// Error read/writing Voltage min warning L1
	Error_Voltage_Guard_Min_Warning_L2: BOOL;	// Error read/writing Voltage min warning L2
	Error_Voltage_Guard_Min_Warning_L3: BOOL;	// Error read/writing Voltage min warning L3
	Error_Voltage_Guard_Max_Warning_L1: BOOL;	// Error read/writing Voltage max warning L1
	Error_Voltage_Guard_Max_Warning_L2: BOOL;	// Error read/writing Voltage max warning L2
	Error_Voltage_Guard_Max_Warning_L3: BOOL;	// Error read/writing Voltage max warning L3
	Error_Voltage_Guard_Max_Error_L1: BOOL;		// Error read/writing Voltage max error L1
	Error_Voltage_Guard_Max_Error_L2: BOOL;		// Error read/writing Voltage max error L2
	Error_Voltage_Guard_Max_Error_L3: BOOL;		// Error read/writing Voltage max error L3

	dummy: INT;
	dummy_bool: bool;
END_VAR

//Case to indicate to the CoE boards FB wich analyzer is selected
CASE GVL_PM_CONFIG.Device_Type_Index OF
	
	0: Device_Type:= 'EL3453';
	
	1: Device_Type:= 'EL3443';
	
	2: Device_Type:= 'EL3783';
	
END_CASE

EL3XXX_Conf(
	NetId_global_assign:= GVL_PM_CONFIG.NetID_EL3XXX, 
	Slave_Add_global_assign:= GVL_PM_CONFIG.SlaveID_EL3XXX,
	NetId_global_assign_2:= GVL_PM_CONFIG.NetID_EL3XXX_2, 
	Slave_Add_global_assign_2:= GVL_PM_CONFIG.SlaveID_EL3XXX_2, 
	EL3_Selection:= Device_Type, 
	Error_selection=> Error_selection, 
	(******************************************************)
	(********************** OUTPUT ************************)
	//Voltage
	Error_Nom_voltage=> Error_Nom_voltage,
	//Frequency
	Error_Nominal_Frequency=> Error_Nominal_Frequency,
	Error_Measurement_freq_range=> Error_Measurement_freq_range,
	//Current trafo
	Error_Current_trafo_rat_L1=> Error_Current_trafo_rat_L1,		
	Error_Current_trafo_rat_L2=> Error_Current_trafo_rat_L2,
	Error_Current_trafo_rat_L3=> Error_Current_trafo_rat_L3,
	//Voltage trafo
	Error_Voltage_trafo_rat_L1=> Error_Voltage_trafo_rat_L1,
	Error_Voltage_trafo_rat_L2=> Error_Voltage_trafo_rat_L2,
	Error_Voltage_trafo_rat_L3=> Error_Voltage_trafo_rat_L3,
	//Current trafo delay
	Error_Current_trafo_dly_L1=> Error_Current_trafo_dly_L1,	
	Error_Current_trafo_dly_L2=> Error_Current_trafo_dly_L2,
	Error_Current_trafo_dly_L3=> Error_Current_trafo_dly_L3,
	//Current trafo for EL3453
	Error_Current_trafo_range_L1=> Error_Current_trafo_range_L1,	
	Error_Current_trafo_range_L2=> Error_Current_trafo_range_L2,
	Error_Current_trafo_range_L3=> Error_Current_trafo_range_L3,
	//Voltage Guard Min Error
	Error_Voltage_Guard_Min_Error_L1=> Error_Voltage_Guard_Min_Error_L1,
	Error_Voltage_Guard_Min_Error_L2=> Error_Voltage_Guard_Min_Error_L2,
	Error_Voltage_Guard_Min_Error_L3=> Error_Voltage_Guard_Min_Error_L3,
	//Voltage Guard Min Warning
	Error_Voltage_Guard_Min_Warning_L1=> Error_Voltage_Guard_Min_Warning_L1,
	Error_Voltage_Guard_Min_Warning_L2=> Error_Voltage_Guard_Min_Warning_L2,
	Error_Voltage_Guard_Min_Warning_L3=> Error_Voltage_Guard_Min_Warning_L3,
	//Voltage Guard Max Warning
	Error_Voltage_Guard_Max_Warning_L1=> Error_Voltage_Guard_Max_Warning_L1,
	Error_Voltage_Guard_Max_Warning_L2=> Error_Voltage_Guard_Max_Warning_L2,
	Error_Voltage_Guard_Max_Warning_L3=> Error_Voltage_Guard_Max_Warning_L3,
	//Voltage Guard Max Error
	Error_Voltage_Guard_Max_Error_L1=> Error_Voltage_Guard_Max_Error_L1,
	Error_Voltage_Guard_Max_Error_L2=> Error_Voltage_Guard_Max_Error_L2,
	Error_Voltage_Guard_Max_Error_L3=> Error_Voltage_Guard_Max_Error_L3,
	(* EL3783 *)
	//Current Range
	Error_Current_Range=> dummy_bool,
	(**********************************************************)
	(********************* SETTINGS INPUTS ********************)
	//Nominal Voltage
	Nominal_Voltage					:= GVL_PM_CONFIG.Nominal_Voltage,
	//Nominal frequency 
	Nominal_Frequency				:= GVL_PM_CONFIG.Nominal_Frequency, 
	Measurement_freq_range			:= GVL_PM_CONFIG.Measurement_freq_range,
	//Current transformers ratio 
	Current_trafo_rat_L1			:= GVL_PM_CONFIG.Current_trafo_rat_L1, 
	Current_trafo_rat_L2			:= GVL_PM_CONFIG.Current_trafo_rat_L2, 
	Current_trafo_rat_L3			:= GVL_PM_CONFIG.Current_trafo_rat_L3,
	//Voltage transformers ratio 
	Voltage_trafo_rat_L1			:= GVL_PM_CONFIG.Voltage_trafo_rat_L1, 
	Voltage_trafo_rat_L2			:= GVL_PM_CONFIG.Voltage_trafo_rat_L2, 
	Voltage_trafo_rat_L3			:= GVL_PM_CONFIG.Voltage_trafo_rat_L3,
	//Current transformers delay 
	Current_trafo_dly_L1			:= GVL_PM_CONFIG.Current_trafo_dly_L1, 
	Current_trafo_dly_L2			:= GVL_PM_CONFIG.Current_trafo_dly_L2, 
	Current_trafo_dly_L3			:= GVL_PM_CONFIG.Current_trafo_dly_L3,
	//Voltage Guard Min Error 
	Voltage_Guard_Min_Error_L1		:= GVL_PM_CONFIG.Voltage_Guard_Min_Error_L1, 
	Voltage_Guard_Min_Error_L2		:= GVL_PM_CONFIG.Voltage_Guard_Min_Error_L2, 
	Voltage_Guard_Min_Error_L3		:= GVL_PM_CONFIG.Voltage_Guard_Min_Error_L3,
	//Voltage Guard Min Warning 
	Voltage_Guard_Min_Warning_L1	:= GVL_PM_CONFIG.Voltage_Guard_Min_Warning_L1, 
	Voltage_Guard_Min_Warning_L2	:= GVL_PM_CONFIG.Voltage_Guard_Min_Warning_L2, 
	Voltage_Guard_Min_Warning_L3	:= GVL_PM_CONFIG.Voltage_Guard_Min_Warning_L3,
	//Voltage Guard Max Warning 
	Voltage_Guard_Max_Warning_L1	:= GVL_PM_CONFIG.Voltage_Guard_Max_Warning_L1, 
	Voltage_Guard_Max_Warning_L2	:= GVL_PM_CONFIG.Voltage_Guard_Max_Warning_L2, 
	Voltage_Guard_Max_Warning_L3	:= GVL_PM_CONFIG.Voltage_Guard_Max_Warning_L3,
	//Voltage Guard Max Error 
	Voltage_Guard_Max_Error_L1		:= GVL_PM_CONFIG.Voltage_Guard_Max_Error_L1, 
	Voltage_Guard_Max_Error_L2		:= GVL_PM_CONFIG.Voltage_Guard_Max_Error_L2, 
	Voltage_Guard_Max_Error_L3		:= GVL_PM_CONFIG.Voltage_Guard_Max_Error_L3,
	(************************* EL3443 *************************)
	//Current transformers ratio for EL3453
	Current_trafo_range_L1			:= GVL_PM_CONFIG.Current_trafo_range_L1, 
	Current_trafo_range_L2			:= GVL_PM_CONFIG.Current_trafo_range_L2, 
	Current_trafo_range_L3			:= GVL_PM_CONFIG.Current_trafo_range_L3,
	(************************* EL3783 *************************)
	//Current Range for EL3783
	Current_Range:= dummy);

END_PROGRAM

// ---- POUs/METERING/METER_EL3453_CFG.TcPOU
FUNCTION_BLOCK METER_EL3453_CFG

VAR_INPUT
	NetId_global_assign : AMSNETID;					// Net Id assignament from the EL3XXX board
	Slave_Add_global_assign : WORD;					// Slave ID address
	NetId_global_assign_2 : AMSNETID;					// Net Id assignament from the EL3XXX board
	Slave_Add_global_assign_2 : WORD;					// Slave ID address
	EL3_Selection : STRING; 						// Selection of power meassurement board: EL3443, EL 3453, EL 3783					
END_VAR


VAR_OUTPUT
	Error_selection : BOOL := TRUE;				// Error in selection of board
	Error_Nom_voltage: BOOL;					// Error read/writing Nominal Voltage
	Error_Nominal_Frequency : BOOL;				// Error read/writing nominal frequency
	Error_Measurement_freq_range : BOOL;		// Error read/writing frequency range working
	Error_Current_trafo_rat_L1 : BOOL;			// Error read/writing Current transformer ratio L1
	Error_Current_trafo_rat_L2 : BOOL;			// Error read/writing Current transformer ratio L2
	Error_Current_trafo_rat_L3 : BOOL;			// Error read/writing Current transformer ratio L3
	Error_Voltage_trafo_rat_L1 : BOOL;			// Error read/writing Voltage transformer ratio L1
	Error_Voltage_trafo_rat_L2 : BOOL;			// Error read/writing Voltage transformer ratio L2
	Error_Voltage_trafo_rat_L3 : BOOL;			// Error read/writing Voltage transformer ratio L3
	Error_Current_trafo_dly_L1 : BOOL;			// Error read/writing Current transformer delay L1	
	Error_Current_trafo_dly_L2 : BOOL;			// Error read/writing Current transformer delay L2
	Error_Current_trafo_dly_L3 : BOOL;			// Error read/writing Current transformer delay L3
	Error_Current_trafo_range_L1 : BOOL;		// Error read/writing Current transformer range L1
	Error_Current_trafo_range_L2 : BOOL;		// Error read/writing Current transformer range L2
	Error_Current_trafo_range_L3 : BOOL;		// Error read/writing Current transformer range L3
	Error_Voltage_Guard_Min_Error_L1 : BOOL;	// Error read/writing Voltage Guard Min Error L1
	Error_Voltage_Guard_Min_Error_L2 : BOOL;	// Error read/writing Voltage Guard Min Error L2
	Error_Voltage_Guard_Min_Error_L3 : BOOL;	// Error read/writing Voltage Guard Min Error L3
	Error_Voltage_Guard_Min_Warning_L1 : BOOL;	// Error read/writing Voltage Guard Min Warning L1
	Error_Voltage_Guard_Min_Warning_L2 : BOOL;	// Error read/writing Voltage Guard Min Warning L2
	Error_Voltage_Guard_Min_Warning_L3 : BOOL;	// Error read/writing Voltage Guard Min Warning L3
	Error_Voltage_Guard_Max_Warning_L1 : BOOL;	// Error read/writing Voltage Guard Max Warning L1
	Error_Voltage_Guard_Max_Warning_L2 : BOOL;	// Error read/writing Voltage Guard Max Warning L2
	Error_Voltage_Guard_Max_Warning_L3 : BOOL;	// Error read/writing Voltage Guard Max Warning L3
	Error_Voltage_Guard_Max_Error_L1 : BOOL;	// Error read/writing Voltage Guard Max Error L1
	Error_Voltage_Guard_Max_Error_L2 : BOOL;	// Error read/writing Voltage Guard Max Error L2
	Error_Voltage_Guard_Max_Error_L3 : BOOL;	// Error read/writing Voltage Guard Max Error L3
	(* EL3783 *)
	Error_Current_Range : BOOL;					// Error read/writing Current Range
END_VAR

VAR_IN_OUT
	
	Nominal_Voltage : REAL;					// Set variable for nominal voltage
	Nominal_Frequency : REAL;				// Set variable for nominal frequency
	Measurement_freq_range : REAL;			// Set variable for frequency range working
	Current_trafo_rat_L1 : REAL;			// Set variable for Current transformer ratio L1
	Current_trafo_rat_L2 : REAL;			// Set variable for Current transformer ratio L2
	Current_trafo_rat_L3 : REAL;			// Set variable for Current transformer ratio L3
	Voltage_trafo_rat_L1 : REAL;			// Set variable for Voltage transformer ratio L1
	Voltage_trafo_rat_L2 : REAL;			// Set variable for Voltage transformer ratio L2
	Voltage_trafo_rat_L3 : REAL;			// Set variable for Voltage transformer ratio L3
	Current_trafo_dly_L1 : REAL;			// Set variable for Current transformer delay L1	
	Current_trafo_dly_L2 : REAL;			// Set variable for Current transformer delay L2
	Current_trafo_dly_L3 : REAL;			// Set variable for Current transformer delay L3
	Current_trafo_range_L1 : UDINT;			// Set variable for Current transformer range L1
	Current_trafo_range_L2 : UDINT;			// Set variable for Current transformer range L2
	Current_trafo_range_L3 : UDINT;			// Set variable for Current transformer range L3
	Voltage_Guard_Min_Error_L1: REAL;		// Set variable for Voltage min error L1
	Voltage_Guard_Min_Error_L2: REAL;		// Set variable for Voltage min error L2
	Voltage_Guard_Min_Error_L3: REAL;		// Set variable for Voltage min error L3
	Voltage_Guard_Min_Warning_L1: REAL;		// Set variable for Voltage min warning L1
	Voltage_Guard_Min_Warning_L2: REAL;		// Set variable for Voltage min warning L2
	Voltage_Guard_Min_Warning_L3: REAL;		// Set variable for Voltage min warning L3
	Voltage_Guard_Max_Warning_L1: REAL;		// Set variable for Voltage max warning L1
	Voltage_Guard_Max_Warning_L2: REAL;		// Set variable for Voltage max warning L2
	Voltage_Guard_Max_Warning_L3: REAL;		// Set variable for Voltage max warning L3
	Voltage_Guard_Max_Error_L1: REAL;		// Set variable for Voltage max error L1
	Voltage_Guard_Max_Error_L2: REAL;		// Set variable for Voltage max error L2
	Voltage_Guard_Max_Error_L3: REAL;		// Set variable for Voltage max error L3
	(* EL3783 *)
	Current_Range : INT;					// Set variable for Current Range EL3783
END_VAR


VAR
	INIT : BOOL := TRUE;					// Launching the initialization of readings	
	INIT_SECOND : BOOL := FALSE;			// It needs to do in three times the init of variables otherwise, the ethercat returns fault
	TRigger_Init_Second : BOOL := TRUE;		// Init to trigger the times
	Delay_second_Init : TON;				// Timer for the second request
	INIT_THIRD : BOOL := FALSE;				// It needs to do in three times the init of variables otherwise, the ethercat returns fault
	TRigger_Init_Third : BOOL := FALSE;		// Init to trigger the times
	Delay_third_Init : TON;					// Timer for the third request

	netID_previous: AMSNETID := [0,0,0,0,0,0];		// Checking if the ID has changed	
	netID_internal: STRING(255);						// Internal ID used for the functions
	netID_previous_2: AMSNETID := [0,0,0,0,0,0];		// Checking if the ID has changed	
	netID_internal_2: STRING(255);						// Internal ID used for the functions		
	i: INT;												// Operand
	
	Exec_Nom_voltage: BOOL;								// Execute command for the writing
	Exec_READ_Nom_voltage: BOOL;						// Execute command for the reading
	Busy_Nom_voltage: BOOL;								// Bus busy will execute the action
	Previous_Nom_voltage_val : REAL;					// Previous value
	
	Exec_Nom_frequency: BOOL;							// Execute command for the writing
	Exec_READ_Nom_frequency: BOOL;						// Execute command for the reading
	Busy_Nom_frequency: BOOL;							// Bus busy will execute the action
	Previous_Nom_frequency_val : REAL;					// Previous value
	
	Exec_Measurement_freq_range: BOOL;					// Execute command for the writing
	Exec_READ_Measurement_freq_range: BOOL;				// Execute command for the reading
	Busy_Measurement_freq_range: BOOL;					// Bus busy will execute the action
	Previous_Measurement_freq_range_val : REAL;			// Previous value
	
	Exec_Current_trafo_rat_L1: BOOL;					// Execute command for the writing
	Exec_READ_Current_trafo_rat_L1: BOOL;				// Execute command for the reading
	Busy_Current_trafo_rat_L1: BOOL;					// Bus busy will execute the action
	Previous_Current_trafo_rat_L1_val : REAL;			// Previous value
	
	Exec_Current_trafo_rat_L2: BOOL;					// Execute command for the writing
	Exec_READ_Current_trafo_rat_L2: BOOL;				// Execute command for the reading
	Busy_Current_trafo_rat_L2: BOOL;					// Bus busy will execute the action
	Previous_Current_trafo_rat_L2_val : REAL;			// Previous value
	
	Exec_Current_trafo_rat_L3: BOOL;					// Execute command for the writing
	Exec_READ_Current_trafo_rat_L3: BOOL;				// Execute command for the reading
	Busy_Current_trafo_rat_L3: BOOL;					// Bus busy will execute the action
	Previous_Current_trafo_rat_L3_val : REAL;			// Previous value
	
	Exec_Voltage_trafo_rat_L1: BOOL;					// Execute command for the writing
	Exec_READ_Voltage_trafo_rat_L1: BOOL;				// Execute command for the reading
	Busy_Voltage_trafo_rat_L1: BOOL;					// Bus busy will execute the action
	Previous_Voltage_trafo_rat_L1_val : REAL;			// Previous value
	
	Exec_Voltage_trafo_rat_L2: BOOL;					// Execute command for the writing
	Exec_READ_Voltage_trafo_rat_L2: BOOL;				// Execute command for the reading
	Busy_Voltage_trafo_rat_L2: BOOL;					// Bus busy will execute the action
	Previous_Voltage_trafo_rat_L2_val : REAL;			// Previous value
	
	Exec_Voltage_trafo_rat_L3: BOOL;					// Execute command for the writing
	Exec_READ_Voltage_trafo_rat_L3: BOOL;				// Execute command for the reading
	Busy_Voltage_trafo_rat_L3: BOOL;					// Bus busy will execute the action
	Previous_Voltage_trafo_rat_L3_val : REAL;			// Previous value
	
	Exec_Current_trafo_dly_L1: BOOL;					// Execute command for the writing
	Exec_READ_Current_trafo_dly_L1: BOOL;				// Execute command for the reading
	Busy_Current_trafo_dly_L1: BOOL;					// Bus busy will execute the action
	Previous_Current_trafo_dly_L1_val : REAL;			// Previous value
	
	Exec_Current_trafo_dly_L2: BOOL;					// Execute command for the writing
	Exec_READ_Current_trafo_dly_L2: BOOL;				// Execute command for the reading
	Busy_Current_trafo_dly_L2: BOOL;					// Bus busy will execute the action
	Previous_Current_trafo_dly_L2_val : REAL;			// Previous value
	
	Exec_Current_trafo_dly_L3: BOOL;					// Execute command for the writing
	Exec_READ_Current_trafo_dly_L3: BOOL;				// Execute command for the reading
	Busy_Current_trafo_dly_L3: BOOL;					// Bus busy will execute the action
	Previous_Current_trafo_dly_L3_val : REAL;			// Previous value
	
	Exec_Current_trafo_range_L1: BOOL;					// Execute command for the writing
	Exec_READ_Current_trafo_range_L1: BOOL;				// Execute command for the reading
	Busy_Current_trafo_range_L1: BOOL;					// Bus busy will execute the action
	Previous_Current_trafo_range_L1_val : UDINT;		// Previous value
	
	Exec_Current_trafo_range_L2: BOOL;					// Execute command for the writing
	Exec_READ_Current_trafo_range_L2: BOOL;				// Execute command for the reading
	Busy_Current_trafo_range_L2: BOOL;					// Bus busy will execute the action
	Previous_Current_trafo_range_L2_val : UDINT;		// Previous value
	
	Exec_Current_trafo_range_L3: BOOL;					// Execute command for the writing
	Exec_READ_Current_trafo_range_L3: BOOL;				// Execute command for the reading
	Busy_Current_trafo_range_L3: BOOL;					// Bus busy will execute the action
	Previous_Current_trafo_range_L3_val : UDINT;		// Previous value
	
	Exec_Voltage_Guard_Min_Error_L1: BOOL;				// Execute command for the writing
	Exec_READ_Voltage_Guard_Min_Error_L1: BOOL;			// Execute command for the reading
	Previous_Voltage_Guard_Min_Error_L1_val : REAL;		// Previous value
	
	Exec_Voltage_Guard_Min_Error_L2: BOOL;				// Execute command for the writing
	Exec_READ_Voltage_Guard_Min_Error_L2: BOOL;			// Execute command for the reading
	Previous_Voltage_Guard_Min_Error_L2_val: REAL;		// Previous value
	
	Exec_Voltage_Guard_Min_Error_L3: BOOL;				// Execute command for the writing
	Exec_READ_Voltage_Guard_Min_Error_L3: BOOL;			// Execute command for the reading
	Previous_Voltage_Guard_Min_Error_L3_val : REAL;		// Previous value
	
	Exec_Voltage_Guard_Min_Warning_L1: BOOL;			// Execute command for the writing
	Exec_READ_Voltage_Guard_Min_Warning_L1: BOOL;		// Execute command for the reading
	Previous_Voltage_Guard_Min_Warning_L1_val : REAL;	// Previous value
	
	Exec_Voltage_Guard_Min_Warning_L2: BOOL;			// Execute command for the writing
	Exec_READ_Voltage_Guard_Min_Warning_L2: BOOL;		// Execute command for the reading
	Previous_Voltage_Guard_Min_Warning_L2_val : REAL;	// Previous value
	
	Exec_Voltage_Guard_Min_Warning_L3: BOOL;			// Execute command for the writing
	Exec_READ_Voltage_Guard_Min_Warning_L3: BOOL;		// Execute command for the reading
	Previous_Voltage_Guard_Min_Warning_L3_val : REAL;	// Previous value
	
	Exec_Voltage_Guard_Max_Warning_L1: BOOL;			// Execute command for the writing
	Exec_READ_Voltage_Guard_Max_Warning_L1: BOOL;		// Execute command for the reading
	Previous_Voltage_Guard_Max_Warning_L1_val : REAL;	// Previous value
	
	Exec_Voltage_Guard_Max_Warning_L2: BOOL;			// Execute command for the writing
	Exec_READ_Voltage_Guard_Max_Warning_L2: BOOL;		// Execute command for the reading
	Previous_Voltage_Guard_Max_Warning_L2_val : REAL;	// Previous value
	
	Exec_Voltage_Guard_Max_Warning_L3: BOOL;			// Execute command for the writing
	Exec_READ_Voltage_Guard_Max_Warning_L3: BOOL;		// Execute command for the reading
	Previous_Voltage_Guard_Max_Warning_L3_val : REAL;	// Previous value
	
	Exec_Voltage_Guard_Max_Error_L1: BOOL;				// Execute command for the writing
	Exec_READ_Voltage_Guard_Max_Error_L1: BOOL;			// Execute command for the reading
	Previous_Voltage_Guard_Max_Error_L1_val : REAL;		// Previous value
	
	Exec_Voltage_Guard_Max_Error_L2: BOOL;				// Execute command for the writing
	Exec_READ_Voltage_Guard_Max_Error_L2: BOOL;			// Execute command for the reading
	Previous_Voltage_Guard_Max_Error_L2_val : REAL;		// Previous value
	
	Exec_Voltage_Guard_Max_Error_L3: BOOL;				// Execute command for the writing
	Exec_READ_Voltage_Guard_Max_Error_L3: BOOL;			// Execute command for the reading
	Previous_Voltage_Guard_Max_Error_L3_val : REAL;		// Previous value
	
	Exec_Current_Range: BOOL;							// Execute command for the writing
	Exec_READ_Current_Range: BOOL;						// Execute command for the reading
	Busy_Current_Range: BOOL;							// Bus busy will execute the action
	Previous_Current_Range_val : INT;					// Previous value
	
	
	Nom_voltage_WR : FB_EcCoESdoWrite;					// Funtion Block writting Nominal voltage 
	Nom_frequency_WR : FB_EcCoESdoWrite;				// Funtion Block writting Nominal frequency 
	Range_freq_WR : FB_EcCoESdoWrite;					// Funtion Block writting Range for frequency 
	Current_trafo_ratio_L1_WR : FB_EcCoESdoWrite;		// Funtion Block writting Current trafo ratio in L1
	Current_trafo_ratio_L2_WR : FB_EcCoESdoWrite;		// Funtion Block writting Current trafo ratio in L2
	Current_trafo_ratio_L3_WR : FB_EcCoESdoWrite;		// Funtion Block writting Current trafo ratio in L3
	Voltage_trafo_ratio_L1_WR : FB_EcCoESdoWrite;		// Funtion Block writting Voltage trafo ratio in L1
	Voltage_trafo_ratio_L2_WR : FB_EcCoESdoWrite;		// Funtion Block writting Voltage trafo ratio in L2
	Voltage_trafo_ratio_L3_WR : FB_EcCoESdoWrite;		// Funtion Block writting Voltage trafo ratio in L3
	Current_trafo_DLY_L1_WR : FB_EcCoESdoWrite;			// Funtion Block writting Current trafo delay in L1
	Current_trafo_DLY_L2_WR : FB_EcCoESdoWrite;			// Funtion Block writting Current trafo delay in L2
	Current_trafo_DLY_L3_WR : FB_EcCoESdoWrite;			// Funtion Block writting Current trafo delay in L3
	Current_trafo_range_L1_WR : FB_EcCoESdoWrite;		// Funtion Block writting Current trafo range in L1
	Current_trafo_range_L2_WR : FB_EcCoESdoWrite;		// Funtion Block writting Current trafo range in L2
	Current_trafo_range_L3_WR : FB_EcCoESdoWrite;		// Funtion Block writting Current trafo range in L3
	Voltage_Guard_Min_Error_L1_WR : FB_EcCoESdoWrite;	// Funtion Block writting Voltage Guard Min Error in L1
	Voltage_Guard_Min_Error_L2_WR : FB_EcCoESdoWrite;	// Funtion Block writting Voltage Guard Min Error in L2
	Voltage_Guard_Min_Error_L3_WR : FB_EcCoESdoWrite;	// Funtion Block writting Voltage Guard Min Error in L3
	Voltage_Guard_Min_Warning_L1_WR : FB_EcCoESdoWrite;	// Funtion Block writting Voltage Guard Min Warning in L1
	Voltage_Guard_Min_Warning_L2_WR : FB_EcCoESdoWrite;	// Funtion Block writting Voltage Guard Min Warning in L2
	Voltage_Guard_Min_Warning_L3_WR : FB_EcCoESdoWrite;	// Funtion Block writting Voltage Guard Min Warning in L3
	Voltage_Guard_Max_Warning_L1_WR : FB_EcCoESdoWrite;	// Funtion Block writting Voltage Guard Max Warning in L1
	Voltage_Guard_Max_Warning_L2_WR : FB_EcCoESdoWrite;	// Funtion Block writting Voltage Guard Max Warning in L2
	Voltage_Guard_Max_Warning_L3_WR : FB_EcCoESdoWrite;	// Funtion Block writting Voltage Guard Max Warning in L3
	Voltage_Guard_Max_Error_L1_WR : FB_EcCoESdoWrite;	// Funtion Block writting Voltage Guard Max Error in L1
	Voltage_Guard_Max_Error_L2_WR : FB_EcCoESdoWrite;	// Funtion Block writting Voltage Guard Max Error in L2
	Voltage_Guard_Max_Error_L3_WR : FB_EcCoESdoWrite;	// Funtion Block writting Voltage Guard Max Error in L3
	Current_Range_WR : FB_EcCoESdoWrite;				// Funtion Block writting Current Range
	
	Nom_voltage_RD : FB_EcCoESdoRead;					// Funtion Block reading Nominal voltage 
	Nom_frequency_RD : FB_EcCoESdoRead;					// Funtion Block reading Nominal frequency 
	Range_freq_RD : FB_EcCoESdoRead;					// Funtion Block reading Range for frequency 
	Current_trafo_ratio_L1_RD : FB_EcCoESdoRead;		// Funtion Block reading Current trafo ratio in L1
	Current_trafo_ratio_L2_RD : FB_EcCoESdoRead;		// Funtion Block reading Current trafo ratio in L2
	Current_trafo_ratio_L3_RD : FB_EcCoESdoRead;		// Funtion Block reading Current trafo ratio in L3
	Voltage_trafo_ratio_L1_RD : FB_EcCoESdoRead;		// Funtion Block reading Voltage trafo ratio in L1
	Voltage_trafo_ratio_L2_RD : FB_EcCoESdoRead;		// Funtion Block reading Voltage trafo ratio in L2
	Voltage_trafo_ratio_L3_RD : FB_EcCoESdoRead;		// Funtion Block reading Voltage trafo ratio in L3
	Current_trafo_DLY_L1_RD : FB_EcCoESdoRead;			// Funtion Block reading Current trafo delay in L1
	Current_trafo_DLY_L2_RD : FB_EcCoESdoRead;			// Funtion Block reading Current trafo delay in L2
	Current_trafo_DLY_L3_RD : FB_EcCoESdoRead;			// Funtion Block reading Current trafo delay in L3
	Current_trafo_range_L1_RD : FB_EcCoESdoRead;		// Funtion Block reading Current trafo range in L1
	Current_trafo_range_L2_RD : FB_EcCoESdoRead;		// Funtion Block reading Current trafo range in L2
	Current_trafo_range_L3_RD : FB_EcCoESdoRead;		// Funtion Block reading Current trafo range in L3
	Voltage_Guard_Min_Error_L1_RD : FB_EcCoESdoRead;	// Funtion Block reading Voltage Guard Min Error in L1
	Voltage_Guard_Min_Error_L2_RD : FB_EcCoESdoRead;	// Funtion Block reading Voltage Guard Min Error in L2
	Voltage_Guard_Min_Error_L3_RD : FB_EcCoESdoRead;	// Funtion Block reading Voltage Guard Min Error in L3
	Voltage_Guard_Min_Warning_L1_RD : FB_EcCoESdoRead;	// Funtion Block reading Voltage Guard Min Warning in L1
	Voltage_Guard_Min_Warning_L2_RD : FB_EcCoESdoRead;	// Funtion Block reading Voltage Guard Min Warning in L2
	Voltage_Guard_Min_Warning_L3_RD : FB_EcCoESdoRead;	// Funtion Block reading Voltage Guard Min Warning in L3
	Voltage_Guard_Max_Warning_L1_RD : FB_EcCoESdoRead;	// Funtion Block reading Voltage Guard Max Warning in L1
	Voltage_Guard_Max_Warning_L2_RD : FB_EcCoESdoRead;	// Funtion Block reading Voltage Guard Max Warning in L2
	Voltage_Guard_Max_Warning_L3_RD : FB_EcCoESdoRead;	// Funtion Block reading Voltage Guard Max Warning in L3
	Voltage_Guard_Max_Error_L1_RD : FB_EcCoESdoRead;	// Funtion Block reading Voltage Guard Max Error in L1
	Voltage_Guard_Max_Error_L2_RD : FB_EcCoESdoRead;	// Funtion Block reading Voltage Guard Max Error in L2
	Voltage_Guard_Max_Error_L3_RD : FB_EcCoESdoRead;	// Funtion Block reading Voltage Guard Max Error in L3
	Current_Range_RD: FB_EcCoESdoRead;					// Funtion Block reading Current Range EL3783
	
	
	Counter_init: INT := 0;
	Counter_init_2: INT := 0;
END_VAR


(************************************************************************************************

							EL3XXX CONFIGURATION FUNCTION BLOCK

*************************************************************************************************

This function block is used to set the parameters up in the EL3XXX power meassurement boards. Here
is set up the following parameters:

- 	Nominal Voltage
- 	Nominal Frequency
- 	Meassurement frequency range
- 	Current transformer ratio L1, L2 and L3
- 	Current delay transformer ratio L1, L2 and L3
- 	Voltage transformer ratio L1, L2 and L3

How must the function be used?

- 	It must be declared 2 variables to be assigned to the AdsAddr of the metering board
- 	The variable netId has format AMSNETID (especial type format for this address, ARRAY [0..5]
- 	The variable port is the slave address and must be declared like a WORD
- 	Each configuration variable is declared as INPUT/OUTPUT so the variables unused must be fulfilled with 
	Dummy variables.
- 	The output variables could be not called
- 	The selection of EL3XXX board can be, EL3443, EL3453 or EL3783. Other declaration reports error
*************************************************************************************************)

(* First of all, it is necessary convert the NetId (AMSNETID) to STRING*)
//IF netID_previous <> NetId_global_assign THEN
	netID_internal := '';
	
	FOR i := 0 TO  5 DO
		
		netID_internal := CONCAT(netID_internal, BYTE_TO_STRING(NetId_global_assign[i]));
			
		IF i < 5 THEN
			netID_internal := CONCAT(netID_internal, '.');
		END_IF
		
	END_FOR
	
	netID_previous := NetId_global_assign;
	
//END_IF	
	
(********************************************* EL3783 ********************************************)

netID_internal_2 := '';
	
	FOR i := 0 TO  5 DO
		
		netID_internal_2 := CONCAT(netID_internal_2, BYTE_TO_STRING(NetId_global_assign_2[i]));
			
		IF i < 5 THEN
			netID_internal_2 := CONCAT(netID_internal_2, '.');
		END_IF
		
	END_FOR
	
	netID_previous_2 := NetId_global_assign_2;	
	

(* It is necessary to know what is the power measurement boards that is going to be configured *)
IF EL3_Selection = 'EL3443' OR EL3_Selection = 'EL3453' THEN
	
	(* In the first scan cycle, the function performs a reading to get the parameters from the board *)
	(* It is necessary send the request in two times, otherwise the last frames reports error*)
	
	IF INIT_SECOND = TRUE THEN	
		IF INIT AND Counter_Init <= 27 THEN
			CASE Counter_init OF
				//Nominal voltage
				0: Exec_READ_Nom_voltage := TRUE;
				//Frequency 
				1: Exec_READ_Nom_frequency := TRUE;
				2: Exec_READ_Measurement_freq_range := TRUE;
				//Current tranformers retio
				3: Exec_READ_Current_trafo_rat_L1 := TRUE;
				4: Exec_READ_Current_trafo_rat_L2 := TRUE;
				5: Exec_READ_Current_trafo_rat_L3 := TRUE;
				//Voltage transformers ratio	
				6: Exec_READ_Voltage_trafo_rat_L1 := TRUE;
				7: Exec_READ_Voltage_trafo_rat_L2 := TRUE;
				8: Exec_READ_Voltage_trafo_rat_L3 := TRUE;
				//Current transformers delay
				9: Exec_READ_Current_trafo_dly_L1 := TRUE;
				10: Exec_READ_Current_trafo_dly_L2 := TRUE;
				11: Exec_READ_Current_trafo_dly_L3 := TRUE;
				//Voltage guard min error
				12: Exec_READ_Voltage_Guard_Min_Error_L1 := TRUE;
				13: Exec_READ_Voltage_Guard_Min_Error_L2 := TRUE;
				14: Exec_READ_Voltage_Guard_Min_Error_L3 := TRUE;
				//Voltage guard min warning
				15: Exec_READ_Voltage_Guard_Min_Warning_L1 := TRUE;
				16: Exec_READ_Voltage_Guard_Min_Warning_L2 := TRUE;
				17: Exec_READ_Voltage_Guard_Min_Warning_L3 := TRUE;
				//Voltage guard max warning
				18: Exec_READ_Voltage_Guard_Max_Warning_L1 := TRUE;
				19: Exec_READ_Voltage_Guard_Max_Warning_L2 := TRUE;
				20: Exec_READ_Voltage_Guard_Max_Warning_L3 := TRUE;
				//Voltage guard max error
				21: Exec_READ_Voltage_Guard_Max_Error_L1 := TRUE;
				22: Exec_READ_Voltage_Guard_Max_Error_L2 := TRUE;
				23: Exec_READ_Voltage_Guard_Max_Error_L3 := TRUE;
				(* EL3453 *)
				//EL3453 current transformers ratios
				24: IF EL3_Selection = 'EL3453' THEN Exec_READ_Current_trafo_range_L1 := TRUE; END_IF
				25: IF EL3_Selection = 'EL3453' THEN Exec_READ_Current_trafo_range_L2 := TRUE; END_IF
				26: IF EL3_Selection = 'EL3453' THEN Exec_READ_Current_trafo_range_L3 := TRUE; END_IF
				
			END_CASE
			Counter_init := Counter_init + 1;
		END_IF
	END_IF

	Delay_second_Init (IN := NOT(INIT_SECOND), PT := T#200MS, Q => INIT_SECOND, ET => );
	
	(* Reset the error selection *)
	Error_selection := FALSE;
	
(***************************************** NOMINAL VOLTAGE *******************************************)
	(* Execution of the writing reading of nominal voltage. When the previous value is diferent to the
	current one, the is executed the command*)
	IF Nominal_Voltage <> Previous_Nom_voltage_val THEN
		Exec_Nom_voltage := TRUE;
	END_IF
	
	(* Function to write the new value in the CoE parameter*)
	Nom_voltage_WR(
		sNetId:= netID_internal, 
		nSlaveAddr:= Slave_Add_global_assign, 
		nSubIndex:= 16#11, 
		nIndex:= 16#F801, 
		pSrcBuf:= ADR(Nominal_Voltage), 
		cbBufLen:= SIZEOF(Nominal_Voltage), 
		bExecute:= Exec_Nom_voltage, 
		tTimeout:= T#1S);
	
	(* Logic to handle the errors and launch the reading*)	
	IF NOT Nom_voltage_WR.bBusy THEN
    	Exec_Nom_voltage := FALSE;
		IF NOT Nom_voltage_WR.bError THEN 
			(* write successful *)
			Error_Nom_voltage := FALSE;
			IF Previous_Nom_voltage_val <> Nominal_Voltage THEN
				Previous_Nom_voltage_val := Nominal_Voltage;
				Exec_READ_Nom_voltage := TRUE;
			END_IF
		ELSE 
			(* write failed *)
			Error_Nom_voltage := Nom_voltage_WR.bError;
			Nominal_Voltage := Previous_Nom_voltage_val;
		END_IF
	
		Nom_voltage_WR(bExecute := FALSE);
	
	END_IF
	
	(* After writting, it is necessary to check if the parameter has been writting correctly *)
	Nom_voltage_RD(
		sNetId:= netID_internal,
		nSlaveAddr := Slave_Add_global_assign, 
		nIndex:= 16#F801, 
		nSubIndex := 16#11, 
		pDstBuf:= ADR(Nominal_Voltage), 
		cbBufLen:=SIZEOF(Nominal_Voltage),
		bExecute:= Exec_READ_Nom_voltage);
	
	(* Logic to handle the errors in the reading *)	
	IF NOT Nom_voltage_RD.bBusy AND NOT Nom_voltage_WR.bBusy THEN
    	Exec_READ_Nom_voltage := FALSE;
		IF NOT Nom_voltage_RD.bError THEN 
			(* write successful *)
			Error_Nom_voltage := FALSE;
			Previous_Nom_voltage_val := Nominal_Voltage;
		ELSE 
			(* write failed *)
			Error_Nom_voltage := Nom_voltage_WR.bError;
    END_IF

    Nom_voltage_RD(bExecute := FALSE);
	
	END_IF
	
(***************************************** NOMINAL VOLTAGE *******************************************)

(***************************************** NOMINAL FREQUENCY *******************************************)
	(* Execution of the writing reading of nominal voltage. When the previous value is diferent to the
	current one, the is executed the command*)
	IF Nominal_Frequency <> Previous_Nom_frequency_val THEN
		Exec_Nom_frequency := TRUE;
	END_IF
	
	(* Function to write the new value in the CoE parameter*)
	Nom_frequency_WR(
		sNetId:= netID_internal, 
		nSlaveAddr:= Slave_Add_global_assign, 
		nSubIndex:= 16#12, 
		nIndex:= 16#F801, 
		pSrcBuf:= ADR(Nominal_Frequency), 
		cbBufLen:= SIZEOF(Nominal_Frequency), 
		bExecute:= Exec_Nom_frequency, 
		tTimeout:= T#1S);
	
	(* Logic to handle the errors and launch the reading*)	
	IF NOT Nom_frequency_WR.bBusy THEN
    	Exec_Nom_frequency := FALSE;
		IF NOT Nom_frequency_WR.bError THEN 
			(* write successful *)
			Error_Nominal_Frequency := FALSE;
			IF Previous_Nom_frequency_val <> Nominal_Frequency THEN
				Previous_Nom_frequency_val := Nominal_Frequency;
				Exec_READ_Nom_frequency := TRUE;
			END_IF
		ELSE 
			(* write failed *)
			Error_Nominal_Frequency := Nom_frequency_WR.bError;
			Nominal_Frequency := Previous_Nom_frequency_val;
		END_IF
	
		Nom_frequency_WR(bExecute := FALSE);
	
	END_IF
	
	(* After writting, it is necessary to check if the parameter has been writting correctly*)
	Nom_frequency_RD(
		sNetId:= netID_internal,
		nSlaveAddr := Slave_Add_global_assign, 
		nIndex:= 16#F801, 
		nSubIndex := 16#12, 
		pDstBuf:= ADR(Nominal_Frequency), 
		cbBufLen:=SIZEOF(Nominal_Frequency),
		bExecute:= Exec_READ_Nom_frequency);
	
	(* Logic to handle the errors in the reading*)	
	IF NOT Nom_frequency_RD.bBusy AND NOT Nom_frequency_WR.bBusy THEN
    	Exec_READ_Nom_frequency := FALSE;
		IF NOT Nom_frequency_RD.bError THEN 
			(* write successful *)
			Error_Nominal_Frequency := FALSE;
			Previous_Nom_frequency_val := Nominal_Frequency;
		ELSE 
			(* write failed *)
			Error_Nominal_Frequency := Nom_frequency_RD.bError;
    END_IF

    Nom_frequency_RD(bExecute := FALSE);
	
	END_IF
	
(***************************************** NOMINAL FREQUENCY *******************************************)

(***************************************** FREQUENCY RANGE *******************************************)
	(* Execution of the writing reading of nominal voltage. When the previous value is diferent to the
	current one, the is executed the command*)
	IF Measurement_freq_range <> Previous_Measurement_freq_range_val THEN
		Exec_Measurement_freq_range := TRUE;
	END_IF
	
	(* Function to write the new value in the CoE parameter*)
	Range_freq_WR(
		sNetId:= netID_internal, 
		nSlaveAddr:= Slave_Add_global_assign, 
		nSubIndex:= 16#12, 
		nIndex:= 16#F800, 
		pSrcBuf:= ADR(Measurement_freq_range), 
		cbBufLen:= SIZEOF(Measurement_freq_range), 
		bExecute:= Exec_Measurement_freq_range, 
		tTimeout:= T#1S);
	
	(* Logic to handle the errors and launch the reading*)	
	IF NOT Range_freq_WR.bBusy THEN
    	Exec_Measurement_freq_range := FALSE;
		IF NOT Range_freq_WR.bError THEN 
			(* write successful *)
			Error_Measurement_freq_range := FALSE;
			IF Previous_Measurement_freq_range_val <> Measurement_freq_range THEN
				Previous_Measurement_freq_range_val := Measurement_freq_range;
				Exec_READ_Measurement_freq_range := TRUE;
			END_IF
		ELSE 
			(* write failed *)
			Error_Measurement_freq_range := Range_freq_WR.bError;
			Measurement_freq_range := Previous_Measurement_freq_range_val;
		END_IF
	
		Range_freq_WR(bExecute := FALSE);
	
	END_IF
	
	(* After writting, it is necessary to check if the parameter has been writting correctly*)
	Range_freq_RD(
		sNetId:= netID_internal,
		nSlaveAddr := Slave_Add_global_assign, 
		nIndex:= 16#F800, 
		nSubIndex := 16#12, 
		pDstBuf:= ADR(Measurement_freq_range), 
		cbBufLen:=SIZEOF(Measurement_freq_range),
		bExecute:= Exec_READ_Measurement_freq_range);
	
	(* Logic to handle the errors in the reading*)	
	IF NOT Range_freq_RD.bBusy AND NOT Range_freq_WR.bBusy THEN
    	Exec_READ_Measurement_freq_range := FALSE;
		IF NOT Range_freq_RD.bError THEN 
			(* write successful *)
			Error_Measurement_freq_range := FALSE;
			Previous_Measurement_freq_range_val := Measurement_freq_range;
		ELSE 
			(* write failed *)
			Error_Measurement_freq_range := Range_freq_RD.bError;
    END_IF

    Range_freq_RD(bExecute := FALSE);
	
	END_IF
	
(***************************************** FREQUENCY RANGE *******************************************)

(********************************** CURRENT TRAFO RATIO L1 *******************************************)
	(* Execution of the writing reading of nominal voltage. When the previous value is diferent to the
	current one, the is executed the command*)
	IF Current_trafo_rat_L1 <> Previous_Current_trafo_rat_L1_val THEN
		Exec_Current_trafo_rat_L1 := TRUE;
	END_IF
	
	(* Function to write the new value in the CoE parameter*)
	Current_trafo_ratio_L1_WR(
		sNetId:= netID_internal, 
		nSlaveAddr:= Slave_Add_global_assign, 
		nSubIndex:= 16#12, 
		nIndex:= 16#8000, 
		pSrcBuf:= ADR(Current_trafo_rat_L1), 
		cbBufLen:= SIZEOF(Current_trafo_rat_L1), 
		bExecute:= Exec_Current_trafo_rat_L1, 
		tTimeout:= T#1S);
	
	(* Logic to handle the errors and launch the reading*)	
	IF NOT Current_trafo_ratio_L1_WR.bBusy THEN
    	Exec_Current_trafo_rat_L1 := FALSE;
		IF NOT Current_trafo_ratio_L1_WR.bError THEN 
			(* write successful *)
			Error_Current_trafo_rat_L1 := FALSE;
			IF Previous_Current_trafo_rat_L1_val <> Current_trafo_rat_L1 THEN
				Previous_Current_trafo_rat_L1_val := Current_trafo_rat_L1;
				Exec_READ_Current_trafo_rat_L1 := TRUE;
			END_IF
		ELSE 
			(* write failed *)
			Error_Current_trafo_rat_L1 := Current_trafo_ratio_L1_WR.bError;
			Current_trafo_rat_L1 := Previous_Current_trafo_rat_L1_val;
		END_IF
	
		Current_trafo_ratio_L1_WR(bExecute := FALSE);
	
	END_IF
	
	(* After writting, it is necessary to check if the parameter has been writting correctly*)
	Current_trafo_ratio_L1_RD(
		sNetId:= netID_internal,
		nSlaveAddr := Slave_Add_global_assign, 
		nIndex:= 16#8000, 
		nSubIndex := 16#12, 
		pDstBuf:= ADR(Current_trafo_rat_L1), 
		cbBufLen:=SIZEOF(Current_trafo_rat_L1),
		bExecute:= Exec_READ_Current_trafo_rat_L1);
	
	(* Logic to handle the errors in the reading*)	
	IF NOT Current_trafo_ratio_L1_RD.bBusy AND NOT Current_trafo_ratio_L1_WR.bBusy THEN
    	Exec_READ_Current_trafo_rat_L1 := FALSE;
		IF NOT Current_trafo_ratio_L1_RD.bError THEN 
			(* write successful *)
			Error_Current_trafo_rat_L1 := FALSE;
			Previous_Current_trafo_rat_L1_val := Current_trafo_rat_L1;
		ELSE 
			(* write failed *)
			Error_Current_trafo_rat_L1 := Current_trafo_ratio_L1_RD.bError;
    END_IF

    Current_trafo_ratio_L1_RD(bExecute := FALSE);
	
	END_IF
	
(********************************** CURRENT TRAFO RATIO L1 *******************************************)
	
(********************************** CURRENT TRAFO RATIO L2 *******************************************)
	(* Execution of the writing reading of nominal voltage. When the previous value is diferent to the
	current one, the is executed the command*)
	IF Current_trafo_rat_L2 <> Previous_Current_trafo_rat_L2_val THEN
		Exec_Current_trafo_rat_L2 := TRUE;
	END_IF
	
	(* Function to write the new value in the CoE parameter*)
	Current_trafo_ratio_L2_WR(
		sNetId:= netID_internal, 
		nSlaveAddr:= Slave_Add_global_assign, 
		nSubIndex:= 16#12, 
		nIndex:= 16#8010, 
		pSrcBuf:= ADR(Current_trafo_rat_L2), 
		cbBufLen:= SIZEOF(Current_trafo_rat_L2), 
		bExecute:= Exec_Current_trafo_rat_L2, 
		tTimeout:= T#1S);
	
	(* Logic to handle the errors and launch the reading*)	
	IF NOT Current_trafo_ratio_L2_WR.bBusy THEN
    	Exec_Current_trafo_rat_L2 := FALSE;
		IF NOT Current_trafo_ratio_L2_WR.bError THEN 
			(* write successful *)
			Error_Current_trafo_rat_L2 := FALSE;
			IF Previous_Current_trafo_rat_L2_val <> Current_trafo_rat_L2 THEN
				Previous_Current_trafo_rat_L2_val := Current_trafo_rat_L2;
				Exec_READ_Current_trafo_rat_L2 := TRUE;
			END_IF
		ELSE 
			(* write failed *)
			Error_Current_trafo_rat_L2 := Current_trafo_ratio_L2_WR.bError;
			Current_trafo_rat_L2 := Previous_Current_trafo_rat_L2_val;
		END_IF
	
		Current_trafo_ratio_L2_WR(bExecute := FALSE);
	
	END_IF
	
	(* After writting, it is necessary to check if the parameter has been writting correctly*)
	Current_trafo_ratio_L2_RD(
		sNetId:= netID_internal,
		nSlaveAddr := Slave_Add_global_assign, 
		nIndex:= 16#8010, 
		nSubIndex := 16#12, 
		pDstBuf:= ADR(Current_trafo_rat_L2), 
		cbBufLen:=SIZEOF(Current_trafo_rat_L2),
		bExecute:= Exec_READ_Current_trafo_rat_L2);
	
	(* Logic to handle the errors in the reading*)	
	IF NOT Current_trafo_ratio_L2_RD.bBusy AND NOT Current_trafo_ratio_L2_WR.bBusy THEN
    	Exec_READ_Current_trafo_rat_L2 := FALSE;
		IF NOT Current_trafo_ratio_L2_RD.bError THEN 
			(* write successful *)
			Error_Current_trafo_rat_L2 := FALSE;
			Previous_Current_trafo_rat_L2_val := Current_trafo_rat_L2;
		ELSE 
			(* write failed *)
			Error_Current_trafo_rat_L2 := Current_trafo_ratio_L2_RD.bError;
    END_IF

    Current_trafo_ratio_L2_RD(bExecute := FALSE);
	
	END_IF
	
(********************************** CURRENT TRAFO RATIO L2 *******************************************)

(********************************** CURRENT TRAFO RATIO L3 *******************************************)
	(* Execution of the writing reading of nominal voltage. When the previous value is diferent to the
	current one, the is executed the command*)
	IF Current_trafo_rat_L3 <> Previous_Current_trafo_rat_L3_val THEN
		Exec_Current_trafo_rat_L3 := TRUE;
	END_IF
	
	(* Function to write the new value in the CoE parameter*)
	Current_trafo_ratio_L3_WR(
		sNetId:= netID_internal, 
		nSlaveAddr:= Slave_Add_global_assign, 
		nSubIndex:= 16#12, 
		nIndex:= 16#8020, 
		pSrcBuf:= ADR(Current_trafo_rat_L3), 
		cbBufLen:= SIZEOF(Current_trafo_rat_L3), 
		bExecute:= Exec_Current_trafo_rat_L3, 
		tTimeout:= T#1S);
	
	(* Logic to handle the errors and launch the reading*)	
	IF NOT Current_trafo_ratio_L3_WR.bBusy THEN
    	Exec_Current_trafo_rat_L3 := FALSE;
		IF NOT Current_trafo_ratio_L3_WR.bError THEN 
			(* write successful *)
			Error_Current_trafo_rat_L3 := FALSE;
			IF Previous_Current_trafo_rat_L3_val <> Current_trafo_rat_L3 THEN
				Previous_Current_trafo_rat_L3_val := Current_trafo_rat_L3;
				Exec_READ_Current_trafo_rat_L3 := TRUE;
			END_IF
		ELSE 
			(* write failed *)
			Error_Current_trafo_rat_L3 := Current_trafo_ratio_L3_WR.bError;
			Current_trafo_rat_L3 := Previous_Current_trafo_rat_L3_val;
		END_IF
	
		Current_trafo_ratio_L3_WR(bExecute := FALSE);
	
	END_IF
	
	(* After writting, it is necessary to check if the parameter has been writting correctly*)
	Current_trafo_ratio_L3_RD(
		sNetId:= netID_internal,
		nSlaveAddr := Slave_Add_global_assign, 
		nIndex:= 16#8020, 
		nSubIndex := 16#12, 
		pDstBuf:= ADR(Current_trafo_rat_L3), 
		cbBufLen:=SIZEOF(Current_trafo_rat_L3),
		bExecute:= Exec_READ_Current_trafo_rat_L3);
	
	(* Logic to handle the errors in the reading*)	
	IF NOT Current_trafo_ratio_L3_RD.bBusy AND NOT Current_trafo_ratio_L3_WR.bBusy THEN
    	Exec_READ_Current_trafo_rat_L3 := FALSE;
		IF NOT Current_trafo_ratio_L3_RD.bError THEN 
			(* write successful *)
			Error_Current_trafo_rat_L3 := FALSE;
			Previous_Current_trafo_rat_L3_val := Current_trafo_rat_L3;
		ELSE 
			(* write failed *)
			Error_Current_trafo_rat_L3 := Current_trafo_ratio_L3_RD.bError;
    END_IF

    Current_trafo_ratio_L3_RD(bExecute := FALSE);
	
	END_IF
	
(********************************** CURRENT TRAFO RATIO L3 *******************************************)

(********************************** VOLTAGE TRAFO RATIO L1 *******************************************)
	(* Execution of the writing reading of nominal voltage. When the previous value is diferent to the
	current one, the is executed the command*)
	IF Voltage_trafo_rat_L1 <> Previous_Voltage_trafo_rat_L1_val THEN
		Exec_Voltage_trafo_rat_L1 := TRUE;
	END_IF
	
	(* Function to write the new value in the CoE parameter*)
	Voltage_trafo_ratio_L1_WR(
		sNetId:= netID_internal, 
		nSlaveAddr:= Slave_Add_global_assign, 
		nSubIndex:= 16#11, 
		nIndex:= 16#8000, 
		pSrcBuf:= ADR(Voltage_trafo_rat_L1), 
		cbBufLen:= SIZEOF(Voltage_trafo_rat_L1), 
		bExecute:= Exec_Voltage_trafo_rat_L1, 
		tTimeout:= T#1S);
	
	(* Logic to handle the errors and launch the reading*)	
	IF NOT Voltage_trafo_ratio_L1_WR.bBusy THEN
    	Exec_Voltage_trafo_rat_L1 := FALSE;
		IF NOT Voltage_trafo_ratio_L1_WR.bError THEN 
			(* write successful *)
			Error_Voltage_trafo_rat_L1 := FALSE;
			IF Previous_Voltage_trafo_rat_L1_val <> Voltage_trafo_rat_L1 THEN
				Previous_Voltage_trafo_rat_L1_val := Voltage_trafo_rat_L1;
				Exec_READ_Voltage_trafo_rat_L1 := TRUE;
			END_IF
		ELSE 
			(* write failed *)
			Error_Voltage_trafo_rat_L1 := Voltage_trafo_ratio_L1_WR.bError;
			Voltage_trafo_rat_L1 := Previous_Voltage_trafo_rat_L1_val;
		END_IF
	
		Voltage_trafo_ratio_L1_WR(bExecute := FALSE);
	
	END_IF
	
	(* After writting, it is necessary to check if the parameter has been writting correctly*)
	Voltage_trafo_ratio_L1_RD(
		sNetId:= netID_internal,
		nSlaveAddr := Slave_Add_global_assign, 
		nIndex:= 16#8000, 
		nSubIndex := 16#11, 
		pDstBuf:= ADR(Voltage_trafo_rat_L1), 
		cbBufLen:=SIZEOF(Voltage_trafo_rat_L1),
		bExecute:= Exec_READ_Voltage_trafo_rat_L1);
	
	(* Logic to handle the errors in the reading*)	
	IF NOT Voltage_trafo_ratio_L1_RD.bBusy AND NOT Voltage_trafo_ratio_L1_WR.bBusy THEN
    	Exec_READ_Voltage_trafo_rat_L1 := FALSE;
		IF NOT Voltage_trafo_ratio_L1_RD.bError THEN 
			(* write successful *)
			Error_Voltage_trafo_rat_L1 := FALSE;
			Previous_Voltage_trafo_rat_L1_val := Voltage_trafo_rat_L1;
		ELSE 
			(* write failed *)
			Error_Voltage_trafo_rat_L1 := Voltage_trafo_ratio_L1_RD.bError;
    END_IF

    Voltage_trafo_ratio_L1_RD(bExecute := FALSE);
	
	END_IF
	
(********************************** VOLTAGE TRAFO RATIO L1 *******************************************)

(********************************** VOLTAGE TRAFO RATIO L2 *******************************************)
	(* Execution of the writing reading of nominal voltage. When the previous value is diferent to the
	current one, the is executed the command*)
	IF Voltage_trafo_rat_L2 <> Previous_Voltage_trafo_rat_L2_val THEN
		Exec_Voltage_trafo_rat_L2 := TRUE;
	END_IF
	
	(* Function to write the new value in the CoE parameter*)
	Voltage_trafo_ratio_L2_WR(
		sNetId:= netID_internal, 
		nSlaveAddr:= Slave_Add_global_assign, 
		nSubIndex:= 16#11, 
		nIndex:= 16#8010, 
		pSrcBuf:= ADR(Voltage_trafo_rat_L2), 
		cbBufLen:= SIZEOF(Voltage_trafo_rat_L2), 
		bExecute:= Exec_Voltage_trafo_rat_L2, 
		tTimeout:= T#1S);
	
	(* Logic to handle the errors and launch the reading*)	
	IF NOT Voltage_trafo_ratio_L2_WR.bBusy THEN
    	Exec_Voltage_trafo_rat_L2 := FALSE;
		IF NOT Voltage_trafo_ratio_L2_WR.bError THEN 
			(* write successful *)
			Error_Voltage_trafo_rat_L2 := FALSE;
			IF Previous_Voltage_trafo_rat_L2_val <> Voltage_trafo_rat_L2 THEN
				Previous_Voltage_trafo_rat_L2_val := Voltage_trafo_rat_L2;
				Exec_READ_Voltage_trafo_rat_L2 := TRUE;
			END_IF
		ELSE 
			(* write failed *)
			Error_Voltage_trafo_rat_L2 := Voltage_trafo_ratio_L2_WR.bError;
			Voltage_trafo_rat_L2 := Previous_Voltage_trafo_rat_L2_val;
		END_IF
	
		Voltage_trafo_ratio_L2_WR(bExecute := FALSE);
	
	END_IF
	
	(* After writting, it is necessary to check if the parameter has been writting correctly*)
	Voltage_trafo_ratio_L2_RD(
		sNetId:= netID_internal,
		nSlaveAddr := Slave_Add_global_assign, 
		nIndex:= 16#8010, 
		nSubIndex := 16#11, 
		pDstBuf:= ADR(Voltage_trafo_rat_L2), 
		cbBufLen:=SIZEOF(Voltage_trafo_rat_L2),
		bExecute:= Exec_READ_Voltage_trafo_rat_L2);
	
	(* Logic to handle the errors in the reading*)	
	IF NOT Voltage_trafo_ratio_L2_RD.bBusy AND NOT Voltage_trafo_ratio_L2_WR.bBusy THEN
    	Exec_READ_Voltage_trafo_rat_L2 := FALSE;
		IF NOT Voltage_trafo_ratio_L2_RD.bError THEN 
			(* write successful *)
			Error_Voltage_trafo_rat_L2 := FALSE;
			Previous_Voltage_trafo_rat_L2_val := Voltage_trafo_rat_L2;
		ELSE 
			(* write failed *)
			Error_Voltage_trafo_rat_L2 := Voltage_trafo_ratio_L2_RD.bError;
    END_IF

    Voltage_trafo_ratio_L2_RD(bExecute := FALSE);
	
	END_IF
	
(********************************** VOLTAGE TRAFO RATIO L2 *******************************************)

(********************************** VOLTAGE TRAFO RATIO L3 *******************************************)
	(* Execution of the writing reading of nominal voltage. When the previous value is diferent to the
	current one, the is executed the command*)
	IF Voltage_trafo_rat_L3 <> Previous_Voltage_trafo_rat_L3_val THEN
		Exec_Voltage_trafo_rat_L3 := TRUE;
	END_IF
	
	(* Function to write the new value in the CoE parameter*)
	Voltage_trafo_ratio_L3_WR(
		sNetId:= netID_internal, 
		nSlaveAddr:= Slave_Add_global_assign, 
		nSubIndex:= 16#11, 
		nIndex:= 16#8020, 
		pSrcBuf:= ADR(Voltage_trafo_rat_L3), 
		cbBufLen:= SIZEOF(Voltage_trafo_rat_L3), 
		bExecute:= Exec_Voltage_trafo_rat_L3, 
		tTimeout:= T#1S);
	
	(* Logic to handle the errors and launch the reading*)	
	IF NOT Voltage_trafo_ratio_L3_WR.bBusy THEN
    	Exec_Voltage_trafo_rat_L3 := FALSE;
		IF NOT Voltage_trafo_ratio_L3_WR.bError THEN 
			(* write successful *)
			Error_Voltage_trafo_rat_L3 := FALSE;
			IF Previous_Voltage_trafo_rat_L3_val <> Voltage_trafo_rat_L3 THEN
				Previous_Voltage_trafo_rat_L3_val := Voltage_trafo_rat_L3;
				Exec_READ_Voltage_trafo_rat_L3 := TRUE;
			END_IF
		ELSE 
			(* write failed *)
			Error_Voltage_trafo_rat_L3 := Voltage_trafo_ratio_L3_WR.bError;
			Voltage_trafo_rat_L3 := Previous_Voltage_trafo_rat_L3_val;
		END_IF
	
		Voltage_trafo_ratio_L3_WR(bExecute := FALSE);
	
	END_IF
	
	(* After writting, it is necessary to check if the parameter has been writting correctly*)
	Voltage_trafo_ratio_L3_RD(
		sNetId:= netID_internal,
		nSlaveAddr := Slave_Add_global_assign, 
		nIndex:= 16#8020, 
		nSubIndex := 16#11, 
		pDstBuf:= ADR(Voltage_trafo_rat_L3), 
		cbBufLen:=SIZEOF(Voltage_trafo_rat_L3),
		bExecute:= Exec_READ_Voltage_trafo_rat_L3);
	
	(* Logic to handle the errors in the reading*)	
	IF NOT Voltage_trafo_ratio_L3_RD.bBusy AND NOT Voltage_trafo_ratio_L3_WR.bBusy THEN
    	Exec_READ_Voltage_trafo_rat_L3 := FALSE;
		IF NOT Voltage_trafo_ratio_L3_RD.bError THEN 
			(* write successful *)
			Error_Voltage_trafo_rat_L3 := FALSE;
			Previous_Voltage_trafo_rat_L3_val := Voltage_trafo_rat_L3;
		ELSE 
			(* write failed *)
			Error_Voltage_trafo_rat_L3 := Voltage_trafo_ratio_L3_RD.bError;
    END_IF

    Voltage_trafo_ratio_L3_RD(bExecute := FALSE);
	
	END_IF
	
(********************************** VOLTAGE TRAFO RATIO L3 *******************************************)

(********************************** CURRENT TRAFO DELAY L1 *******************************************)
	(* Execution of the writing reading of nominal voltage. When the previous value is diferent to the
	current one, the is executed the command*)
	IF Current_trafo_dly_L1 <> Previous_Current_trafo_dly_L1_val THEN
		Exec_Current_trafo_dly_L1 := TRUE;
	END_IF
	
	(* Function to write the new value in the CoE parameter*)
	Current_trafo_dly_L1_WR(
		sNetId:= netID_internal, 
		nSlaveAddr:= Slave_Add_global_assign, 
		nSubIndex:= 16#13, 
		nIndex:= 16#8000, 
		pSrcBuf:= ADR(Current_trafo_dly_L1), 
		cbBufLen:= SIZEOF(Current_trafo_dly_L1), 
		bExecute:= Exec_Current_trafo_dly_L1, 
		tTimeout:= T#1S);
	
	(* Logic to handle the errors and launch the reading*)	
	IF NOT Current_trafo_dly_L1_WR.bBusy THEN
    	Exec_Current_trafo_dly_L1 := FALSE;
		IF NOT Current_trafo_dly_L1_WR.bError THEN 
			(* write successful *)
			Error_Current_trafo_dly_L1 := FALSE;
			IF Previous_Current_trafo_dly_L1_val <> Current_trafo_dly_L1 THEN
				Previous_Current_trafo_dly_L1_val := Current_trafo_dly_L1;
				Exec_READ_Current_trafo_dly_L1 := TRUE;
			END_IF
		ELSE 
			(* write failed *)
			Error_Current_trafo_dly_L1 := Current_trafo_dly_L1_WR.bError;
			Current_trafo_dly_L1 := Previous_Current_trafo_dly_L1_val;
		END_IF
	
		Current_trafo_dly_L1_WR(bExecute := FALSE);
	
	END_IF
	
	(* After writting, it is necessary to check if the parameter has been writting correctly*)
	Current_trafo_dly_L1_RD(
		sNetId:= netID_internal,
		nSlaveAddr := Slave_Add_global_assign, 
		nIndex:= 16#8000, 
		nSubIndex := 16#13, 
		pDstBuf:= ADR(Current_trafo_dly_L1), 
		cbBufLen:=SIZEOF(Current_trafo_dly_L1),
		bExecute:= Exec_READ_Current_trafo_dly_L1);
	
	(* Logic to handle the errors in the reading*)	
	IF NOT Current_trafo_dly_L1_RD.bBusy AND NOT Current_trafo_dly_L1_WR.bBusy THEN
    	Exec_READ_Current_trafo_dly_L1 := FALSE;
		IF NOT Current_trafo_dly_L1_RD.bError THEN 
			(* write successful *)
			Error_Current_trafo_dly_L1 := FALSE;
			Previous_Current_trafo_dly_L1_val := Current_trafo_dly_L1;
		ELSE 
			(* write failed *)
			Error_Current_trafo_dly_L1 := Current_trafo_dly_L1_RD.bError;
    END_IF

    Current_trafo_dly_L1_RD(bExecute := FALSE);
	
	END_IF
	
(********************************** CURRENT TRAFO DELAY L1 *******************************************)

(********************************** CURRENT TRAFO DELAY L2 *******************************************)
	(* Execution of the writing reading of nominal voltage. When the previous value is diferent to the
	current one, the is executed the command*)
	IF Current_trafo_dly_L2 <> Previous_Current_trafo_dly_L2_val THEN
		Exec_Current_trafo_dly_L2 := TRUE;
	END_IF
	
	(* Function to write the new value in the CoE parameter*)
	Current_trafo_dly_L2_WR(
		sNetId:= netID_internal, 
		nSlaveAddr:= Slave_Add_global_assign, 
		nSubIndex:= 16#13, 
		nIndex:= 16#8010, 
		pSrcBuf:= ADR(Current_trafo_dly_L2), 
		cbBufLen:= SIZEOF(Current_trafo_dly_L2), 
		bExecute:= Exec_Current_trafo_dly_L2, 
		tTimeout:= T#1S);
	
	(* Logic to handle the errors and launch the reading*)	
	IF NOT Current_trafo_dly_L2_WR.bBusy THEN
    	Exec_Current_trafo_dly_L2 := FALSE;
		IF NOT Current_trafo_dly_L2_WR.bError THEN 
			(* write successful *)
			Error_Current_trafo_dly_L2 := FALSE;
			IF Previous_Current_trafo_dly_L2_val <> Current_trafo_dly_L2 THEN
				Previous_Current_trafo_dly_L2_val := Current_trafo_dly_L2;
				Exec_READ_Current_trafo_dly_L2 := TRUE;
			END_IF
		ELSE 
			(* write failed *)
			Error_Current_trafo_dly_L2 := Current_trafo_dly_L2_WR.bError;
			Current_trafo_dly_L2 := Previous_Current_trafo_dly_L2_val;
		END_IF
	
		Current_trafo_dly_L2_WR(bExecute := FALSE);
	
	END_IF
	
	(* After writting, it is necessary to check if the parameter has been writting correctly*)
	Current_trafo_dly_L2_RD(
		sNetId:= netID_internal,
		nSlaveAddr := Slave_Add_global_assign, 
		nIndex:= 16#8010, 
		nSubIndex := 16#13, 
		pDstBuf:= ADR(Current_trafo_dly_L2), 
		cbBufLen:=SIZEOF(Current_trafo_dly_L2),
		bExecute:= Exec_READ_Current_trafo_dly_L2);
	
	(* Logic to handle the errors in the reading*)	
	IF NOT Current_trafo_dly_L2_RD.bBusy AND NOT Current_trafo_dly_L2_WR.bBusy THEN
    	Exec_READ_Current_trafo_dly_L2 := FALSE;
		IF NOT Current_trafo_dly_L2_RD.bError THEN 
			(* write successful *)
			Error_Current_trafo_dly_L2 := FALSE;
			Previous_Current_trafo_dly_L2_val := Current_trafo_dly_L2;
		ELSE 
			(* write failed *)
			Error_Current_trafo_dly_L2 := Current_trafo_dly_L2_RD.bError;
    END_IF

    Current_trafo_dly_L2_RD(bExecute := FALSE);
	
	END_IF
	
(********************************** CURRENT TRAFO DELAY L2 *******************************************)

(********************************** CURRENT TRAFO DELAY L3 *******************************************)
	(* Execution of the writing reading of nominal voltage. When the previous value is diferent to the
	current one, the is executed the command*)
	IF Current_trafo_dly_L3 <> Previous_Current_trafo_dly_L3_val THEN
		Exec_Current_trafo_dly_L3 := TRUE;
	END_IF
	
	(* Function to write the new value in the CoE parameter*)
	Current_trafo_dly_L3_WR(
		sNetId:= netID_internal, 
		nSlaveAddr:= Slave_Add_global_assign, 
		nSubIndex:= 16#13, 
		nIndex:= 16#8020, 
		pSrcBuf:= ADR(Current_trafo_dly_L3), 
		cbBufLen:= SIZEOF(Current_trafo_dly_L3), 
		bExecute:= Exec_Current_trafo_dly_L3, 
		tTimeout:= T#1S);
	
	(* Logic to handle the errors and launch the reading*)	
	IF NOT Current_trafo_dly_L3_WR.bBusy THEN
    	Exec_Current_trafo_dly_L3 := FALSE;
		IF NOT Current_trafo_dly_L3_WR.bError THEN 
			(* write successful *)
			Error_Current_trafo_dly_L3 := FALSE;
			IF Previous_Current_trafo_dly_L3_val <> Current_trafo_dly_L3 THEN
				Previous_Current_trafo_dly_L3_val := Current_trafo_dly_L3;
				Exec_READ_Current_trafo_dly_L3 := TRUE;
			END_IF
		ELSE 
			(* write failed *)
			Error_Current_trafo_dly_L3 := Current_trafo_dly_L3_WR.bError;
			Current_trafo_dly_L3 := Previous_Current_trafo_dly_L3_val;
		END_IF
	
		Current_trafo_dly_L3_WR(bExecute := FALSE);
	
	END_IF
	
	(* After writting, it is necessary to check if the parameter has been writting correctly*)
	Current_trafo_dly_L3_RD(
		sNetId:= netID_internal,
		nSlaveAddr := Slave_Add_global_assign, 
		nIndex:= 16#8020, 
		nSubIndex := 16#13, 
		pDstBuf:= ADR(Current_trafo_dly_L3), 
		cbBufLen:=SIZEOF(Current_trafo_dly_L3),
		bExecute:= Exec_READ_Current_trafo_dly_L3);
	
	(* Logic to handle the errors in the reading*)	
	IF NOT Current_trafo_dly_L3_RD.bBusy AND NOT Current_trafo_dly_L3_WR.bBusy THEN
    	Exec_READ_Current_trafo_dly_L3 := FALSE;
		IF NOT Current_trafo_dly_L3_RD.bError THEN 
			(* write successful *)
			Error_Current_trafo_dly_L3 := FALSE;
			Previous_Current_trafo_dly_L3_val := Current_trafo_dly_L3;
		ELSE 
			(* write failed *)
			Error_Current_trafo_dly_L3 := Current_trafo_dly_L3_RD.bError;
    END_IF

    Current_trafo_dly_L3_RD(bExecute := FALSE);
	
	END_IF
	
(********************************** CURRENT TRAFO DELAY L3 *******************************************)

(********************************* VOLTAGE GUARD MIN ERROR L1 ****************************************)
	(* Execution of the writing reading of Voltage Guard Min Error L1. When the previous value is diferent to the
	current one, the is executed the command*)
	IF Voltage_Guard_Min_Error_L1 <> Previous_Voltage_Guard_Min_Error_L1_val THEN
		Exec_Voltage_Guard_Min_Error_L1 := TRUE;
	END_IF
	
	(* Function to write the new value in the CoE parameter*)
	Voltage_Guard_Min_Error_L1_WR(
		sNetId:= netID_internal, 
		nSlaveAddr:= Slave_Add_global_assign, 
		nSubIndex:= 16#11, 
		nIndex:= 16#8001, 
		pSrcBuf:= ADR(Voltage_Guard_Min_Error_L1), 
		cbBufLen:= SIZEOF(Voltage_Guard_Min_Error_L1), 
		bExecute:= Exec_Voltage_Guard_Min_Error_L1, 
		tTimeout:= T#1S);
	
	(* Logic to handle the errors and launch the reading*)	
	IF NOT Voltage_Guard_Min_Error_L1_WR.bBusy THEN
    	Exec_Voltage_Guard_Min_Error_L1 := FALSE;
		IF NOT Voltage_Guard_Min_Error_L1_WR.bError THEN 
			(* write successful *)
			Error_Voltage_Guard_Min_Error_L1 := FALSE;
			IF Previous_Voltage_Guard_Min_Error_L1_val <> Voltage_Guard_Min_Error_L1 THEN
				Previous_Voltage_Guard_Min_Error_L1_val := Voltage_Guard_Min_Error_L1;
				Exec_READ_Voltage_Guard_Min_Error_L1 := TRUE;
			END_IF
		ELSE 
			(* write failed *)
			Error_Voltage_Guard_Min_Error_L1 := Voltage_Guard_Min_Error_L1_WR.bError;
			Voltage_Guard_Min_Error_L1 := Previous_Voltage_Guard_Min_Error_L1_val;
		END_IF
	
		Voltage_Guard_Min_Error_L1_WR(bExecute := FALSE);
	
	END_IF
	
